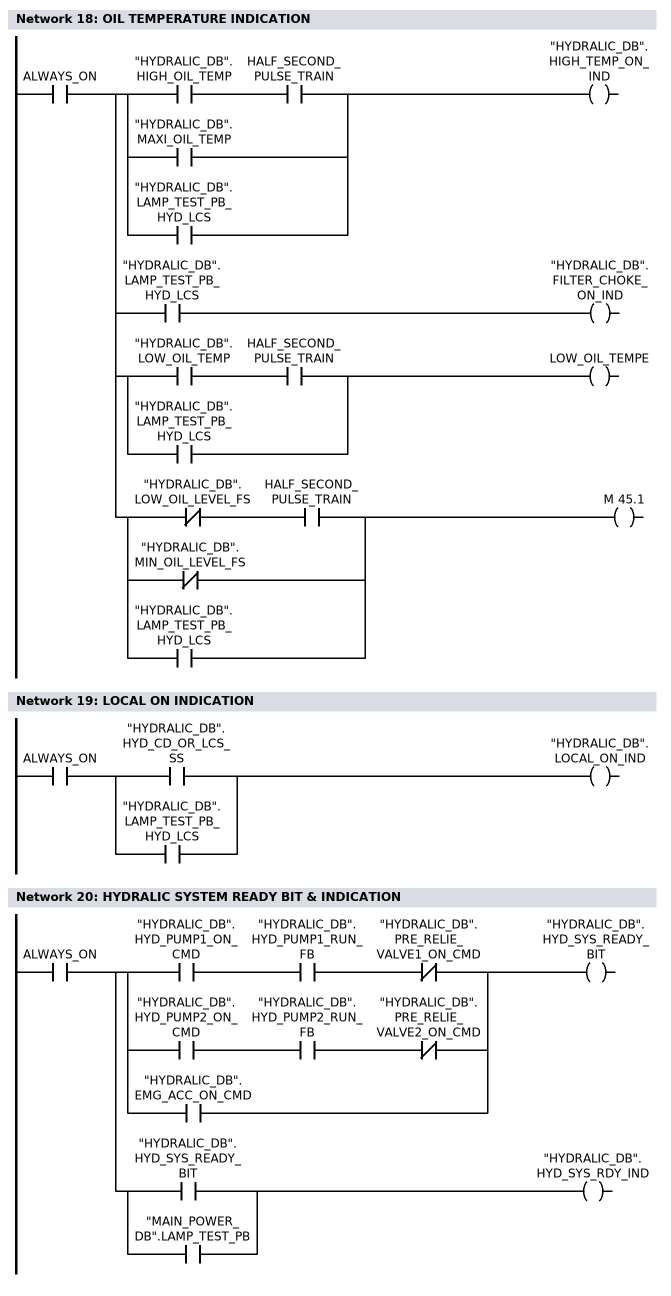
[picture p48: HYDRALIC_FUNCTION networks 18-20]
NETWORK
TITLE = OIL TEMPERATURE INDICATION
      A     "ALWAYS_ON";
      =     L 0.0;
      A     L 0.0;
      A(;
      A     "HYDRALIC_DB".HIGH_OIL_TEMP;
      A     "HALF_SECOND_PULSE_TRAIN";
      O     "HYDRALIC_DB".MAXI_OIL_TEMP;
      O     "HYDRALIC_DB".LAMP_TEST_PB_HYD_LCS;
      );
      =     "HYDRALIC_DB".HIGH_TEMP_ON_IND;
      A     L 0.0;
      A     "HYDRALIC_DB".LAMP_TEST_PB_HYD_LCS;
      =     "HYDRALIC_DB".FILTER_CHOKE_ON_IND;
      A     L 0.0;
      A(;
      A     "HYDRALIC_DB".LOW_OIL_TEMP;
      A     "HALF_SECOND_PULSE_TRAIN";
      O     "HYDRALIC_DB".LAMP_TEST_PB_HYD_LCS;
      );
      =     "LOW_OIL_TEMPE";
      A     L 0.0;
      A(;
      AN    "HYDRALIC_DB".LOW_OIL_LEVEL_FS;
      A     "HALF_SECOND_PULSE_TRAIN";
      ON    "HYDRALIC_DB".MIN_OIL_LEVEL_FS;
      O     "HYDRALIC_DB".LAMP_TEST_PB_HYD_LCS;
      );
      =     M 45.1;
NETWORK
TITLE = LOCAL ON INDICATION
      A     "ALWAYS_ON";
      A(;
      O     "HYDRALIC_DB".HYD_CD_OR_LCS_SS;
      O     "HYDRALIC_DB".LAMP_TEST_PB_HYD_LCS;
      );
      =     "HYDRALIC_DB".LOCAL_ON_IND;
NETWORK
TITLE = HYDRALIC SYSTEM READY BIT & INDICATION
      A     "ALWAYS_ON";
      =     L 0.0;
      A     L 0.0;
      A(;
      A     "HYDRALIC_DB".HYD_PUMP1_ON_CMD;
      A     "HYDRALIC_DB".HYD_PUMP1_RUN_FB;
      AN    "HYDRALIC_DB".PRE_RELIE_VALVE1_ON_CMD;
      O;
      A     "HYDRALIC_DB".HYD_PUMP2_ON_CMD;
      A     "HYDRALIC_DB".HYD_PUMP2_RUN_FB;
      AN    "HYDRALIC_DB".PRE_RELIE_VALVE2_ON_CMD;
      O     "HYDRALIC_DB".EMG_ACC_ON_CMD;
      );
      =     "HYDRALIC_DB".HYD_SYS_READY_BIT;
      A     L 0.0;
      A(;
      O     "HYDRALIC_DB".HYD_SYS_READY_BIT;
      O     "MAIN_POWER_DB".LAMP_TEST_PB;
      );
      =     "HYDRALIC_DB".HYD_SYS_RDY_IND;
END_FUNCTION

FUNCTION "TRAVEL_DRIVE" : VOID	// FC 8
AUTHOR : Arun_Ram
VERSION : 0.1
BEGIN
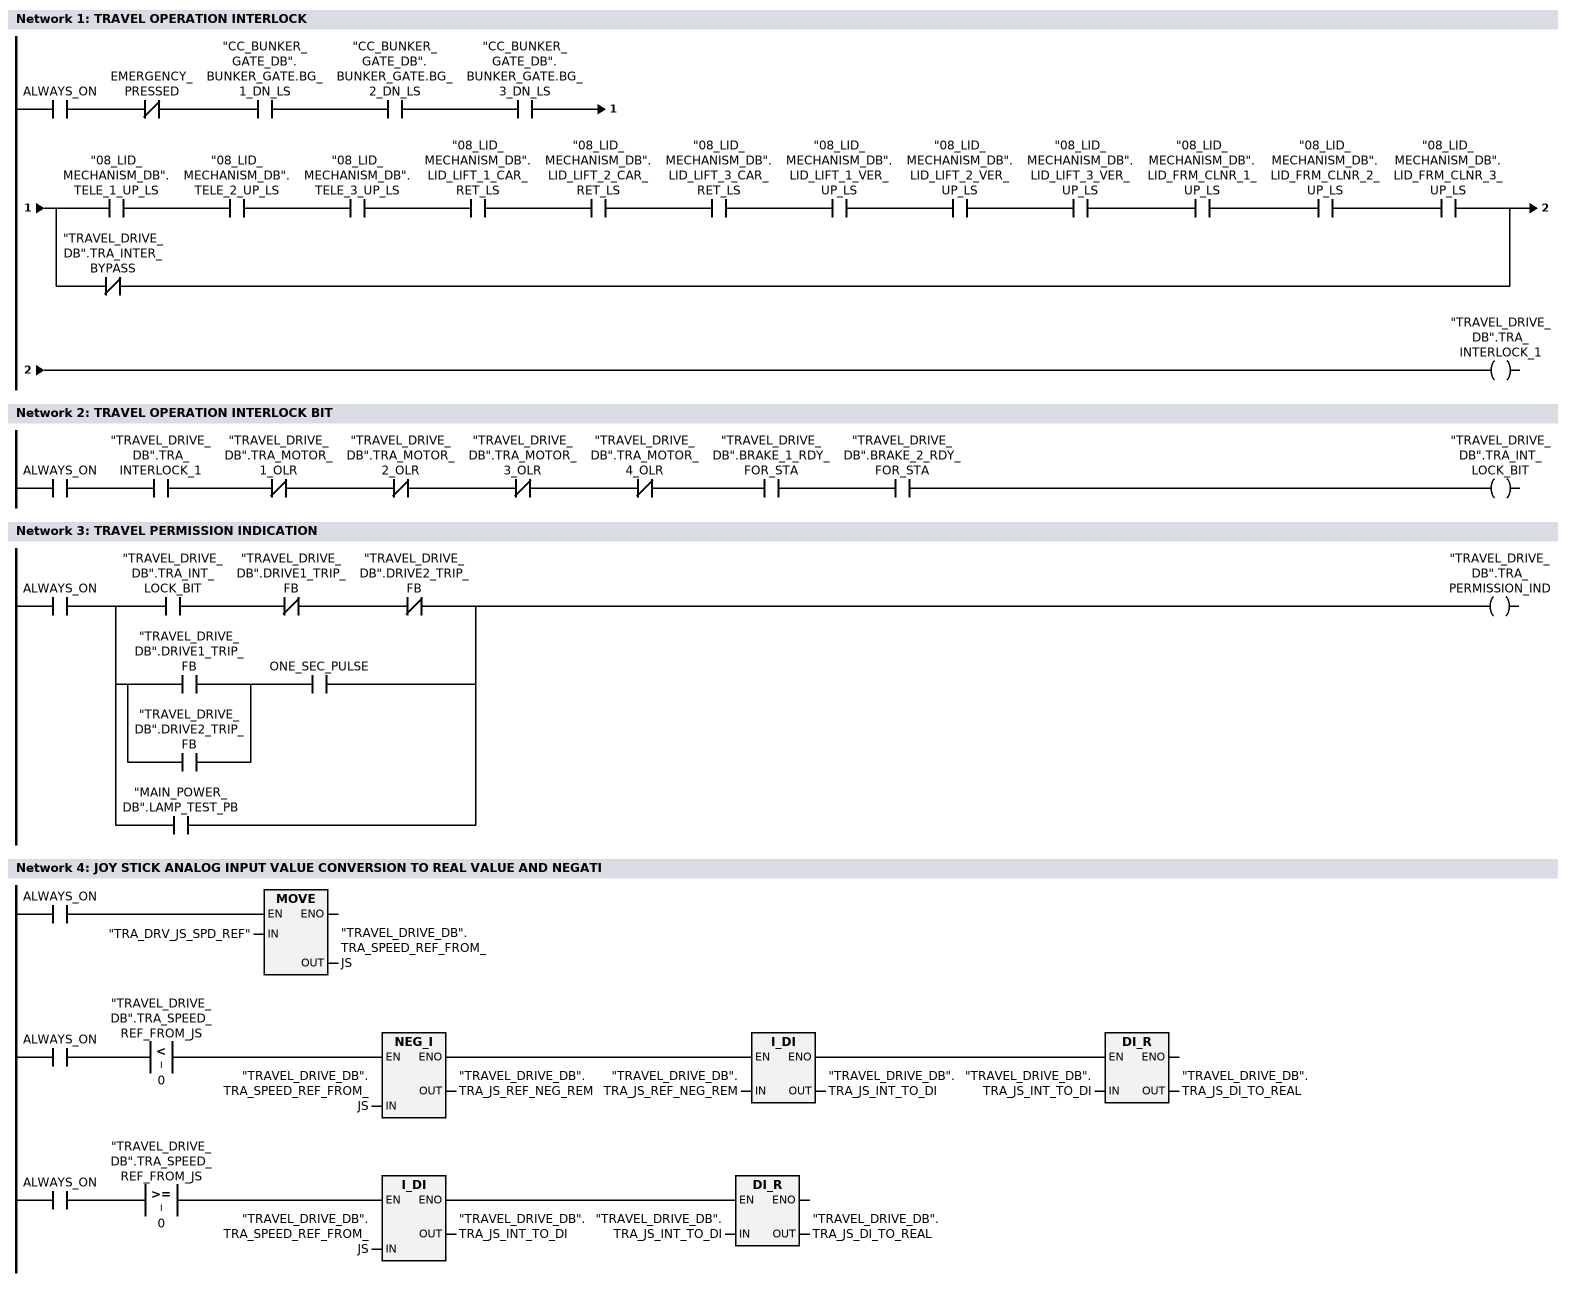
NETWORK
TITLE = TRAVEL OPERATION INTERLOCK
      A     "ALWAYS_ON";
      AN    "EMERGENCY_PRESSED";
      A     "CC_BUNKER_GATE_DB".BUNKER_GATE.BG_1_DN_LS;
      A     "CC_BUNKER_GATE_DB".BUNKER_GATE.BG_2_DN_LS;
      A     "CC_BUNKER_GATE_DB".BUNKER_GATE.BG_3_DN_LS;
      A(;
      A     "08_LID_MECHANISM_DB".TELE_1_UP_LS;
      A     "08_LID_MECHANISM_DB".TELE_2_UP_LS;
      A     "08_LID_MECHANISM_DB".TELE_3_UP_LS;
      A     "08_LID_MECHANISM_DB".LID_LIFT_1_CAR_RET_LS;
      A     "08_LID_MECHANISM_DB".LID_LIFT_2_CAR_RET_LS;
      A     "08_LID_MECHANISM_DB".LID_LIFT_3_CAR_RET_LS;
      A     "08_LID_MECHANISM_DB".LID_LIFT_1_VER_UP_LS;
      A     "08_LID_MECHANISM_DB".LID_LIFT_2_VER_UP_LS;
      A     "08_LID_MECHANISM_DB".LID_LIFT_3_VER_UP_LS;
      A     "08_LID_MECHANISM_DB".LID_FRM_CLNR_1_UP_LS;
      A     "08_LID_MECHANISM_DB".LID_FRM_CLNR_2_UP_LS;
      A     "08_LID_MECHANISM_DB".LID_FRM_CLNR_3_UP_LS;
      ON    "TRAVEL_DRIVE_DB".TRA_INTER_BYPASS;
      );
      =     "TRAVEL_DRIVE_DB".TRA_INTERLOCK_1;
NETWORK
TITLE = TRAVEL OPERATION INTERLOCK BIT
      A     "ALWAYS_ON";
      A     "TRAVEL_DRIVE_DB".TRA_INTERLOCK_1;
      AN    "TRAVEL_DRIVE_DB".TRA_MOTOR_1_OLR;
      AN    "TRAVEL_DRIVE_DB".TRA_MOTOR_2_OLR;
      AN    "TRAVEL_DRIVE_DB".TRA_MOTOR_3_OLR;
      AN    "TRAVEL_DRIVE_DB".TRA_MOTOR_4_OLR;
      A     "TRAVEL_DRIVE_DB".BRAKE_1_RDY_FOR_STA;
      A     "TRAVEL_DRIVE_DB".BRAKE_2_RDY_FOR_STA;
      =     "TRAVEL_DRIVE_DB".TRA_INT_LOCK_BIT;
NETWORK
TITLE = TRAVEL PERMISSION INDICATION
      A     "ALWAYS_ON";
      A(;
      A     "TRAVEL_DRIVE_DB".TRA_INT_LOCK_BIT;
      AN    "TRAVEL_DRIVE_DB".DRIVE1_TRIP_FB;
      AN    "TRAVEL_DRIVE_DB".DRIVE2_TRIP_FB;
      O;
      A(;
      O     "TRAVEL_DRIVE_DB".DRIVE1_TRIP_FB;
      O     "TRAVEL_DRIVE_DB".DRIVE2_TRIP_FB;
      );
      A     "ONE_SEC_PULSE";
      O     "MAIN_POWER_DB".LAMP_TEST_PB;
      );
      =     "TRAVEL_DRIVE_DB".TRA_PERMISSION_IND;
NETWORK
TITLE = JOY STICK ANALOG INPUT VALUE CONVERSION TO REAL VALUE AND NEGATI
//JOY STICK ANALOG INPUT VALUE CONVERTION TO REAL VALUE AND NEGATIVE TO POSITIVE 
//CONVERTION
      A     "ALWAYS_ON";
      =     L 0.0;
      A     L 0.0;
      JNB   _001;
      L     "TRA_DRV_JS_SPD_REF";
      T     "TRAVEL_DRIVE_DB".TRA_SPEED_REF_FROM_JS;
_001: NOP   0;
      A(;
      A(;
      A     L 0.0;
      A(;
      L     "TRAVEL_DRIVE_DB".TRA_SPEED_REF_FROM_JS;
      L     0;
      <I;
      );
      JNB   _002;
      L     "TRAVEL_DRIVE_DB".TRA_SPEED_REF_FROM_JS;
      NEGI;
      T     "TRAVEL_DRIVE_DB".TRA_JS_REF_NEG_REM;
      AN    OV;
      SAVE;
      CLR;
_002: A     BR;
      );
      JNB   _003;
      L     "TRAVEL_DRIVE_DB".TRA_JS_REF_NEG_REM;
      ITD;
      T     "TRAVEL_DRIVE_DB".TRA_JS_INT_TO_DI;
      SET;
      SAVE;
      CLR;
_003: A     BR;
      );
      JNB   _004;
      L     "TRAVEL_DRIVE_DB".TRA_JS_INT_TO_DI;
      DTR;
      T     "TRAVEL_DRIVE_DB".TRA_JS_DI_TO_REAL;
_004: NOP   0;
      A(;
      A     L 0.0;
      A(;
      L     "TRAVEL_DRIVE_DB".TRA_SPEED_REF_FROM_JS;
      L     0;
      >=I;
      );
      JNB   _005;
      L     "TRAVEL_DRIVE_DB".TRA_SPEED_REF_FROM_JS;
      ITD;
      T     "TRAVEL_DRIVE_DB".TRA_JS_INT_TO_DI;
      SET;
      SAVE;
      CLR;
_005: A     BR;
      );
      JNB   _006;
      L     "TRAVEL_DRIVE_DB".TRA_JS_INT_TO_DI;
      DTR;
      T     "TRAVEL_DRIVE_DB".TRA_JS_DI_TO_REAL;
_006: NOP   0;
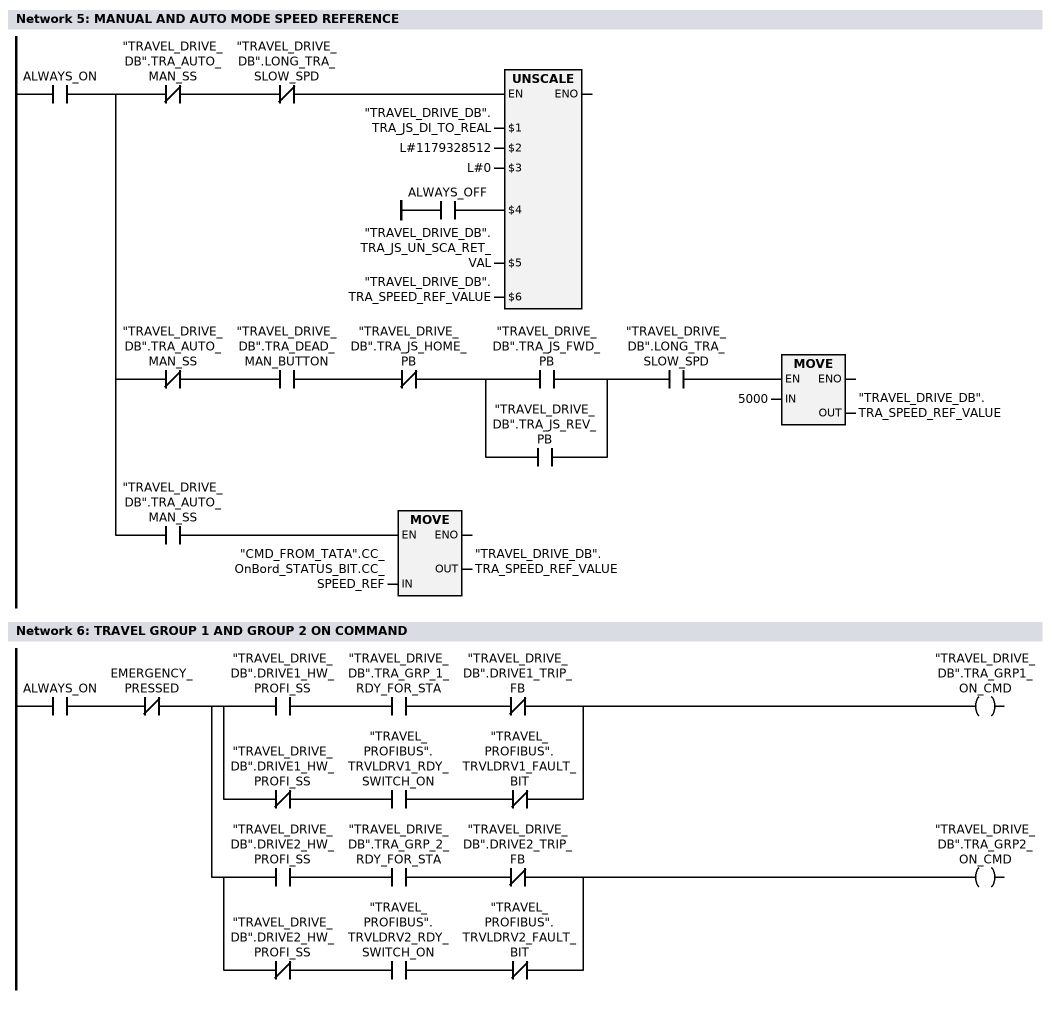
NETWORK
TITLE = MANUAL AND AUTO MODE SPEED REFERENCE
//JOY STICK ANALOG INPUT VALUE SCALLING WITH UNSCALLING BLOCK IN MANUAL MODE AND
//PROFIBUS SPEED REFERENCE VALUE TRANSFER IN AUTO MODE
//
      A     "ALWAYS_ON";
      =     L 0.0;
      A     "ALWAYS_OFF";
      =     L 0.1;
      BLD   103;
      A     L 0.0;
      AN    "TRAVEL_DRIVE_DB".TRA_AUTO_MAN_SS;
      AN    "TRAVEL_DRIVE_DB".LONG_TRA_SLOW_SPD;
      JNB   _007;
      CALL  "UNSCALE" (
           $1                       := "TRAVEL_DRIVE_DB".TRA_JS_DI_TO_REAL,
           $2                       := L#1179328512,
           $3                       := L#0,
           $4                       := L 0.1,
           $5                       := "TRAVEL_DRIVE_DB".TRA_JS_UN_SCA_RET_VAL,
           $6                       := "TRAVEL_DRIVE_DB".TRA_SPEED_REF_VALUE);
_007: NOP   0;
      A     L 0.0;
      AN    "TRAVEL_DRIVE_DB".TRA_AUTO_MAN_SS;
      A     "TRAVEL_DRIVE_DB".TRA_DEAD_MAN_BUTTON;
      AN    "TRAVEL_DRIVE_DB".TRA_JS_HOME_PB;
      A(;
      O     "TRAVEL_DRIVE_DB".TRA_JS_FWD_PB;
      O     "TRAVEL_DRIVE_DB".TRA_JS_REV_PB;
      );
      A     "TRAVEL_DRIVE_DB".LONG_TRA_SLOW_SPD;
      JNB   _008;
      L     5000;
      T     "TRAVEL_DRIVE_DB".TRA_SPEED_REF_VALUE;
_008: NOP   0;
      A     L 0.0;
      A     "TRAVEL_DRIVE_DB".TRA_AUTO_MAN_SS;
      JNB   _009;
      L     "CMD_FROM_TATA".CC_OnBord_STATUS_BIT.CC_SPEED_REF;
      T     "TRAVEL_DRIVE_DB".TRA_SPEED_REF_VALUE;
_009: NOP   0;
NETWORK
TITLE = TRAVEL GROUP 1 AND GROUP 2 ON COMMAND
      A     "ALWAYS_ON";
      AN    "EMERGENCY_PRESSED";
      =     L 0.0;
      A     L 0.0;
      A(;
      A     "TRAVEL_DRIVE_DB".DRIVE1_HW_PROFI_SS;
      A     "TRAVEL_DRIVE_DB".TRA_GRP_1_RDY_FOR_STA;
      AN    "TRAVEL_DRIVE_DB".DRIVE1_TRIP_FB;
      O;
      AN    "TRAVEL_DRIVE_DB".DRIVE1_HW_PROFI_SS;
      A     "TRAVEL_PROFIBUS".TRVLDRV1_RDY_SWITCH_ON;
      AN    "TRAVEL_PROFIBUS".TRVLDRV1_FAULT_BIT;
      );
      =     "TRAVEL_DRIVE_DB".TRA_GRP1_ON_CMD;
      A     L 0.0;
      A(;
      A     "TRAVEL_DRIVE_DB".DRIVE2_HW_PROFI_SS;
      A     "TRAVEL_DRIVE_DB".TRA_GRP_2_RDY_FOR_STA;
      AN    "TRAVEL_DRIVE_DB".DRIVE2_TRIP_FB;
      O;
      AN    "TRAVEL_DRIVE_DB".DRIVE2_HW_PROFI_SS;
      A     "TRAVEL_PROFIBUS".TRVLDRV2_RDY_SWITCH_ON;
      AN    "TRAVEL_PROFIBUS".TRVLDRV2_FAULT_BIT;
      );
      =     "TRAVEL_DRIVE_DB".TRA_GRP2_ON_CMD;
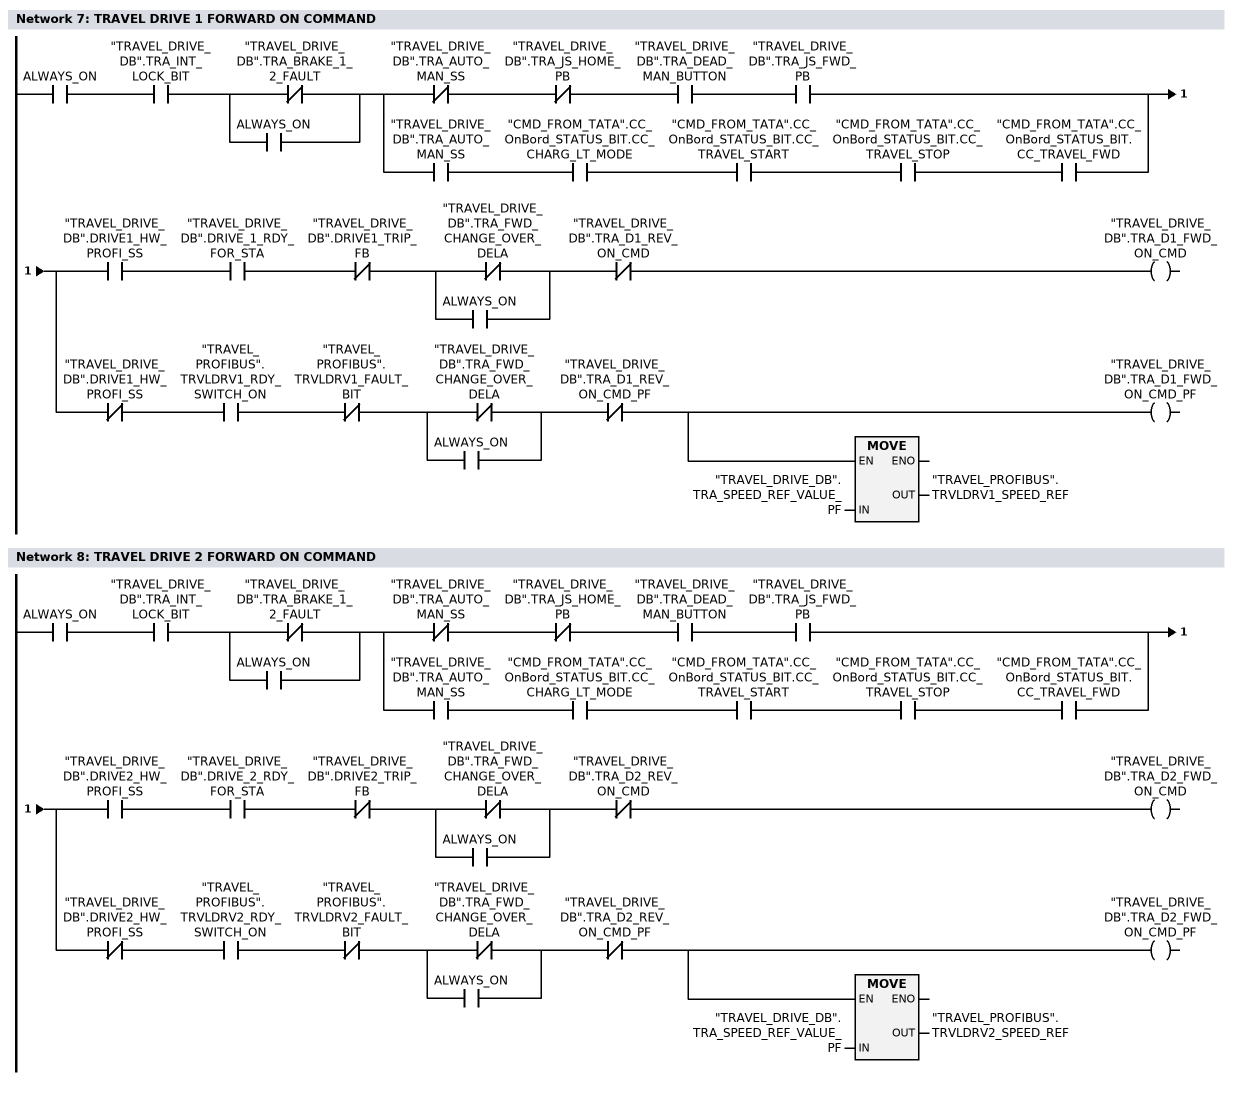
NETWORK
TITLE = TRAVEL DRIVE 1 FORWARD ON COMMAND
      A     "ALWAYS_ON";
      A     "TRAVEL_DRIVE_DB".TRA_INT_LOCK_BIT;
      A(;
      ON    "TRAVEL_DRIVE_DB".TRA_BRAKE_1_2_FAULT;
      O     "ALWAYS_ON";
      );
      A(;
      AN    "TRAVEL_DRIVE_DB".TRA_AUTO_MAN_SS;
      AN    "TRAVEL_DRIVE_DB".TRA_JS_HOME_PB;
      A     "TRAVEL_DRIVE_DB".TRA_DEAD_MAN_BUTTON;
      A     "TRAVEL_DRIVE_DB".TRA_JS_FWD_PB;
      O;
      A     "TRAVEL_DRIVE_DB".TRA_AUTO_MAN_SS;
      A     "CMD_FROM_TATA".CC_OnBord_STATUS_BIT.CC_CHARG_LT_MODE;
      A     "CMD_FROM_TATA".CC_OnBord_STATUS_BIT.CC_TRAVEL_START;
      A     "CMD_FROM_TATA".CC_OnBord_STATUS_BIT.CC_TRAVEL_STOP;
      A     "CMD_FROM_TATA".CC_OnBord_STATUS_BIT.CC_TRAVEL_FWD;
      );
      =     L 0.0;
      A     L 0.0;
      A     "TRAVEL_DRIVE_DB".DRIVE1_HW_PROFI_SS;
      A     "TRAVEL_DRIVE_DB".DRIVE_1_RDY_FOR_STA;
      AN    "TRAVEL_DRIVE_DB".DRIVE1_TRIP_FB;
      A(;
      ON    "TRAVEL_DRIVE_DB".TRA_FWD_CHANGE_OVER_DELA;
      O     "ALWAYS_ON";
      );
      AN    "TRAVEL_DRIVE_DB".TRA_D1_REV_ON_CMD;
      =     "TRAVEL_DRIVE_DB".TRA_D1_FWD_ON_CMD;
      A     L 0.0;
      AN    "TRAVEL_DRIVE_DB".DRIVE1_HW_PROFI_SS;
      A     "TRAVEL_PROFIBUS".TRVLDRV1_RDY_SWITCH_ON;
      AN    "TRAVEL_PROFIBUS".TRVLDRV1_FAULT_BIT;
      A(;
      ON    "TRAVEL_DRIVE_DB".TRA_FWD_CHANGE_OVER_DELA;
      O     "ALWAYS_ON";
      );
      AN    "TRAVEL_DRIVE_DB".TRA_D1_REV_ON_CMD_PF;
      =     L 0.1;
      A     L 0.1;
      BLD   102;
      =     "TRAVEL_DRIVE_DB".TRA_D1_FWD_ON_CMD_PF;
      A     L 0.1;
      JNB   _00a;
      L     "TRAVEL_DRIVE_DB".TRA_SPEED_REF_VALUE_PF;
      T     "TRAVEL_PROFIBUS".TRVLDRV1_SPEED_REF;
_00a: NOP   0;
NETWORK
TITLE = TRAVEL DRIVE 2 FORWARD ON COMMAND
      A     "ALWAYS_ON";
      A     "TRAVEL_DRIVE_DB".TRA_INT_LOCK_BIT;
      A(;
      ON    "TRAVEL_DRIVE_DB".TRA_BRAKE_1_2_FAULT;
      O     "ALWAYS_ON";
      );
      A(;
      AN    "TRAVEL_DRIVE_DB".TRA_AUTO_MAN_SS;
      AN    "TRAVEL_DRIVE_DB".TRA_JS_HOME_PB;
      A     "TRAVEL_DRIVE_DB".TRA_DEAD_MAN_BUTTON;
      A     "TRAVEL_DRIVE_DB".TRA_JS_FWD_PB;
      O;
      A     "TRAVEL_DRIVE_DB".TRA_AUTO_MAN_SS;
      A     "CMD_FROM_TATA".CC_OnBord_STATUS_BIT.CC_CHARG_LT_MODE;
      A     "CMD_FROM_TATA".CC_OnBord_STATUS_BIT.CC_TRAVEL_START;
      A     "CMD_FROM_TATA".CC_OnBord_STATUS_BIT.CC_TRAVEL_STOP;
      A     "CMD_FROM_TATA".CC_OnBord_STATUS_BIT.CC_TRAVEL_FWD;
      );
      =     L 0.0;
      A     L 0.0;
      A     "TRAVEL_DRIVE_DB".DRIVE2_HW_PROFI_SS;
      A     "TRAVEL_DRIVE_DB".DRIVE_2_RDY_FOR_STA;
      AN    "TRAVEL_DRIVE_DB".DRIVE2_TRIP_FB;
      A(;
      ON    "TRAVEL_DRIVE_DB".TRA_FWD_CHANGE_OVER_DELA;
      O     "ALWAYS_ON";
      );
      AN    "TRAVEL_DRIVE_DB".TRA_D2_REV_ON_CMD;
      =     "TRAVEL_DRIVE_DB".TRA_D2_FWD_ON_CMD;
      A     L 0.0;
      AN    "TRAVEL_DRIVE_DB".DRIVE2_HW_PROFI_SS;
      A     "TRAVEL_PROFIBUS".TRVLDRV2_RDY_SWITCH_ON;
      AN    "TRAVEL_PROFIBUS".TRVLDRV2_FAULT_BIT;
      A(;
      ON    "TRAVEL_DRIVE_DB".TRA_FWD_CHANGE_OVER_DELA;
      O     "ALWAYS_ON";
      );
      AN    "TRAVEL_DRIVE_DB".TRA_D2_REV_ON_CMD_PF;
      =     L 0.1;
      A     L 0.1;
      BLD   102;
      =     "TRAVEL_DRIVE_DB".TRA_D2_FWD_ON_CMD_PF;
      A     L 0.1;
      JNB   _00b;
      L     "TRAVEL_DRIVE_DB".TRA_SPEED_REF_VALUE_PF;
      T     "TRAVEL_PROFIBUS".TRVLDRV2_SPEED_REF;
_00b: NOP   0;
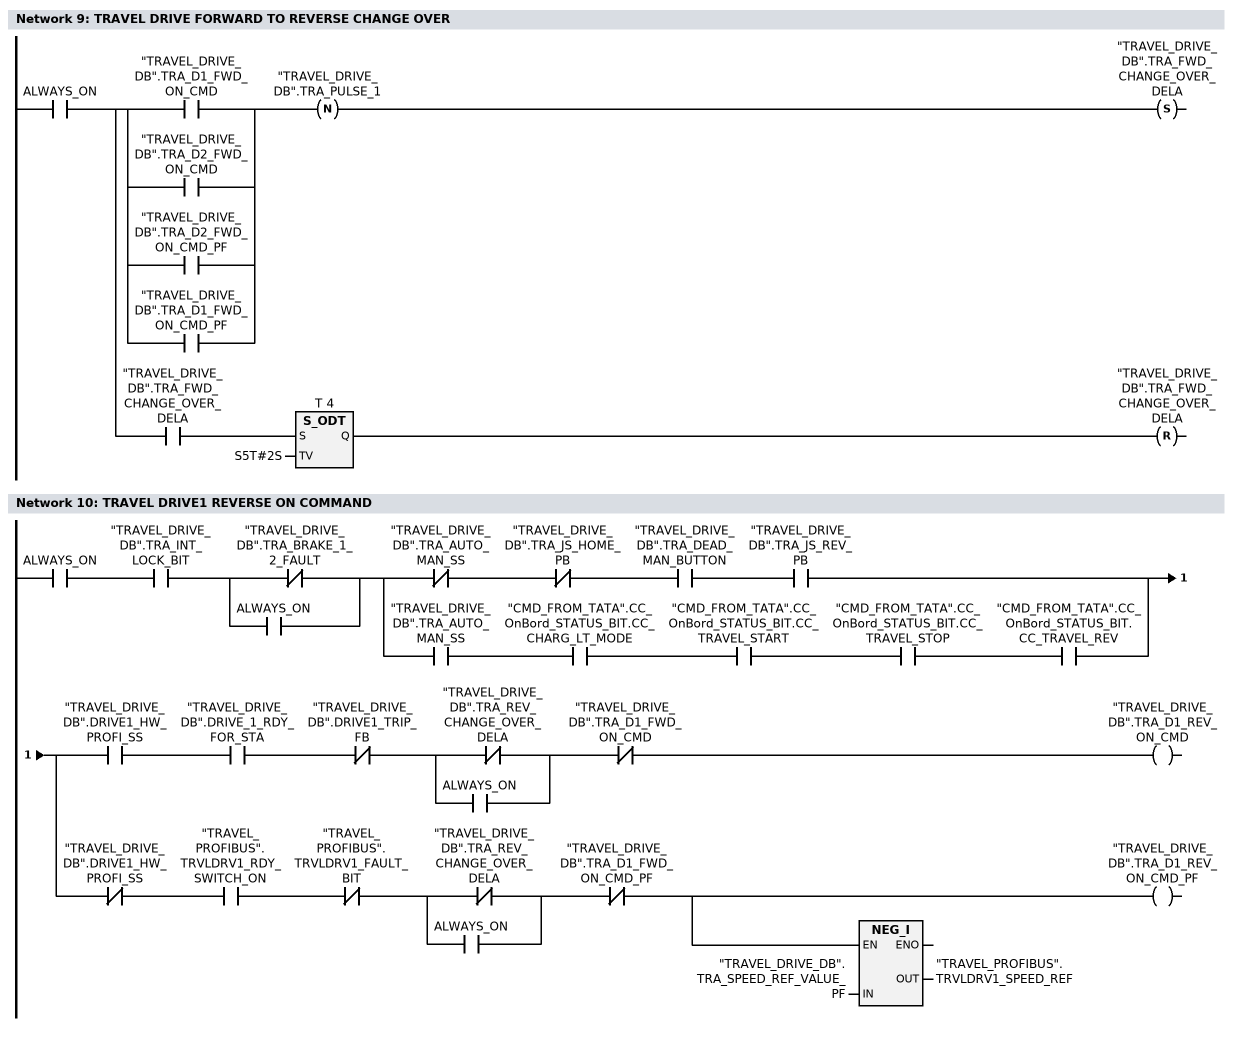
NETWORK
TITLE = TRAVEL DRIVE FORWARD TO REVERSE CHANGE OVER
      A     "ALWAYS_ON";
      =     L 0.0;
      A     L 0.0;
      A(;
      O     "TRAVEL_DRIVE_DB".TRA_D1_FWD_ON_CMD;
      O     "TRAVEL_DRIVE_DB".TRA_D2_FWD_ON_CMD;
      O     "TRAVEL_DRIVE_DB".TRA_D2_FWD_ON_CMD_PF;
      O     "TRAVEL_DRIVE_DB".TRA_D1_FWD_ON_CMD_PF;
      );
      FN    "TRAVEL_DRIVE_DB".TRA_PULSE_1;
      S     "TRAVEL_DRIVE_DB".TRA_FWD_CHANGE_OVER_DELA;
      A     L 0.0;
      A     "TRAVEL_DRIVE_DB".TRA_FWD_CHANGE_OVER_DELA;
      L     S5T#2S;
      SD    T 4;
      NOP   0;
      NOP   0;
      NOP   0;
      A     T 4;
      R     "TRAVEL_DRIVE_DB".TRA_FWD_CHANGE_OVER_DELA;
NETWORK
TITLE = TRAVEL DRIVE1 REVERSE ON COMMAND
      A     "ALWAYS_ON";
      A     "TRAVEL_DRIVE_DB".TRA_INT_LOCK_BIT;
      A(;
      ON    "TRAVEL_DRIVE_DB".TRA_BRAKE_1_2_FAULT;
      O     "ALWAYS_ON";
      );
      A(;
      AN    "TRAVEL_DRIVE_DB".TRA_AUTO_MAN_SS;
      AN    "TRAVEL_DRIVE_DB".TRA_JS_HOME_PB;
      A     "TRAVEL_DRIVE_DB".TRA_DEAD_MAN_BUTTON;
      A     "TRAVEL_DRIVE_DB".TRA_JS_REV_PB;
      O;
      A     "TRAVEL_DRIVE_DB".TRA_AUTO_MAN_SS;
      A     "CMD_FROM_TATA".CC_OnBord_STATUS_BIT.CC_CHARG_LT_MODE;
      A     "CMD_FROM_TATA".CC_OnBord_STATUS_BIT.CC_TRAVEL_START;
      A     "CMD_FROM_TATA".CC_OnBord_STATUS_BIT.CC_TRAVEL_STOP;
      A     "CMD_FROM_TATA".CC_OnBord_STATUS_BIT.CC_TRAVEL_REV;
      );
      =     L 0.0;
      A     L 0.0;
      A     "TRAVEL_DRIVE_DB".DRIVE1_HW_PROFI_SS;
      A     "TRAVEL_DRIVE_DB".DRIVE_1_RDY_FOR_STA;
      AN    "TRAVEL_DRIVE_DB".DRIVE1_TRIP_FB;
      A(;
      ON    "TRAVEL_DRIVE_DB".TRA_REV_CHANGE_OVER_DELA;
      O     "ALWAYS_ON";
      );
      AN    "TRAVEL_DRIVE_DB".TRA_D1_FWD_ON_CMD;
      =     "TRAVEL_DRIVE_DB".TRA_D1_REV_ON_CMD;
      A     L 0.0;
      AN    "TRAVEL_DRIVE_DB".DRIVE1_HW_PROFI_SS;
      A     "TRAVEL_PROFIBUS".TRVLDRV1_RDY_SWITCH_ON;
      AN    "TRAVEL_PROFIBUS".TRVLDRV1_FAULT_BIT;
      A(;
      ON    "TRAVEL_DRIVE_DB".TRA_REV_CHANGE_OVER_DELA;
      O     "ALWAYS_ON";
      );
      AN    "TRAVEL_DRIVE_DB".TRA_D1_FWD_ON_CMD_PF;
      =     L 0.1;
      A     L 0.1;
      BLD   102;
      =     "TRAVEL_DRIVE_DB".TRA_D1_REV_ON_CMD_PF;
      A     L 0.1;
      JNB   _00c;
      L     "TRAVEL_DRIVE_DB".TRA_SPEED_REF_VALUE_PF;
      NEGI;
      T     "TRAVEL_PROFIBUS".TRVLDRV1_SPEED_REF;
_00c: NOP   0;
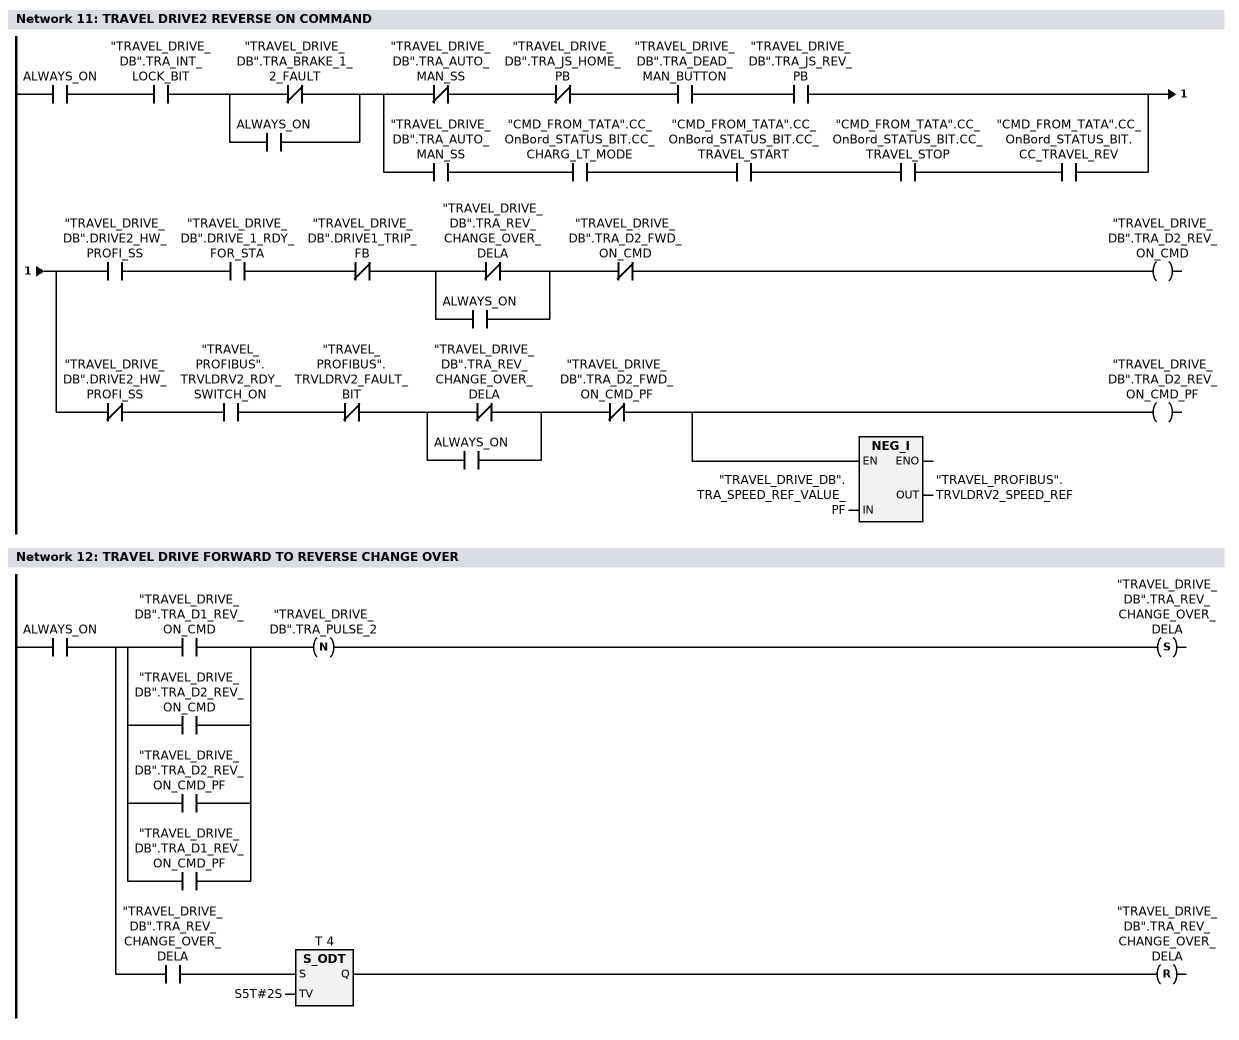
NETWORK
TITLE = TRAVEL DRIVE2 REVERSE ON COMMAND
      A     "ALWAYS_ON";
      A     "TRAVEL_DRIVE_DB".TRA_INT_LOCK_BIT;
      A(;
      ON    "TRAVEL_DRIVE_DB".TRA_BRAKE_1_2_FAULT;
      O     "ALWAYS_ON";
      );
      A(;
      AN    "TRAVEL_DRIVE_DB".TRA_AUTO_MAN_SS;
      AN    "TRAVEL_DRIVE_DB".TRA_JS_HOME_PB;
      A     "TRAVEL_DRIVE_DB".TRA_DEAD_MAN_BUTTON;
      A     "TRAVEL_DRIVE_DB".TRA_JS_REV_PB;
      O;
      A     "TRAVEL_DRIVE_DB".TRA_AUTO_MAN_SS;
      A     "CMD_FROM_TATA".CC_OnBord_STATUS_BIT.CC_CHARG_LT_MODE;
      A     "CMD_FROM_TATA".CC_OnBord_STATUS_BIT.CC_TRAVEL_START;
      A     "CMD_FROM_TATA".CC_OnBord_STATUS_BIT.CC_TRAVEL_STOP;
      A     "CMD_FROM_TATA".CC_OnBord_STATUS_BIT.CC_TRAVEL_REV;
      );
      =     L 0.0;
      A     L 0.0;
      A     "TRAVEL_DRIVE_DB".DRIVE2_HW_PROFI_SS;
      A     "TRAVEL_DRIVE_DB".DRIVE_1_RDY_FOR_STA;
      AN    "TRAVEL_DRIVE_DB".DRIVE1_TRIP_FB;
      A(;
      ON    "TRAVEL_DRIVE_DB".TRA_REV_CHANGE_OVER_DELA;
      O     "ALWAYS_ON";
      );
      AN    "TRAVEL_DRIVE_DB".TRA_D2_FWD_ON_CMD;
      =     "TRAVEL_DRIVE_DB".TRA_D2_REV_ON_CMD;
      A     L 0.0;
      AN    "TRAVEL_DRIVE_DB".DRIVE2_HW_PROFI_SS;
      A     "TRAVEL_PROFIBUS".TRVLDRV2_RDY_SWITCH_ON;
      AN    "TRAVEL_PROFIBUS".TRVLDRV2_FAULT_BIT;
      A(;
      ON    "TRAVEL_DRIVE_DB".TRA_REV_CHANGE_OVER_DELA;
      O     "ALWAYS_ON";
      );
      AN    "TRAVEL_DRIVE_DB".TRA_D2_FWD_ON_CMD_PF;
      =     L 0.1;
      A     L 0.1;
      BLD   102;
      =     "TRAVEL_DRIVE_DB".TRA_D2_REV_ON_CMD_PF;
      A     L 0.1;
      JNB   _00d;
      L     "TRAVEL_DRIVE_DB".TRA_SPEED_REF_VALUE_PF;
      NEGI;
      T     "TRAVEL_PROFIBUS".TRVLDRV2_SPEED_REF;
_00d: NOP   0;
NETWORK
TITLE = TRAVEL DRIVE FORWARD TO REVERSE CHANGE OVER
      A     "ALWAYS_ON";
      =     L 0.0;
      A     L 0.0;
      A(;
      O     "TRAVEL_DRIVE_DB".TRA_D1_REV_ON_CMD;
      O     "TRAVEL_DRIVE_DB".TRA_D2_REV_ON_CMD;
      O     "TRAVEL_DRIVE_DB".TRA_D2_REV_ON_CMD_PF;
      O     "TRAVEL_DRIVE_DB".TRA_D1_REV_ON_CMD_PF;
      );
      FN    "TRAVEL_DRIVE_DB".TRA_PULSE_2;
      S     "TRAVEL_DRIVE_DB".TRA_REV_CHANGE_OVER_DELA;
      A     L 0.0;
      A     "TRAVEL_DRIVE_DB".TRA_REV_CHANGE_OVER_DELA;
      L     S5T#2S;
      SD    T 4;
      NOP   0;
      NOP   0;
      NOP   0;
      A     T 4;
      R     "TRAVEL_DRIVE_DB".TRA_REV_CHANGE_OVER_DELA;
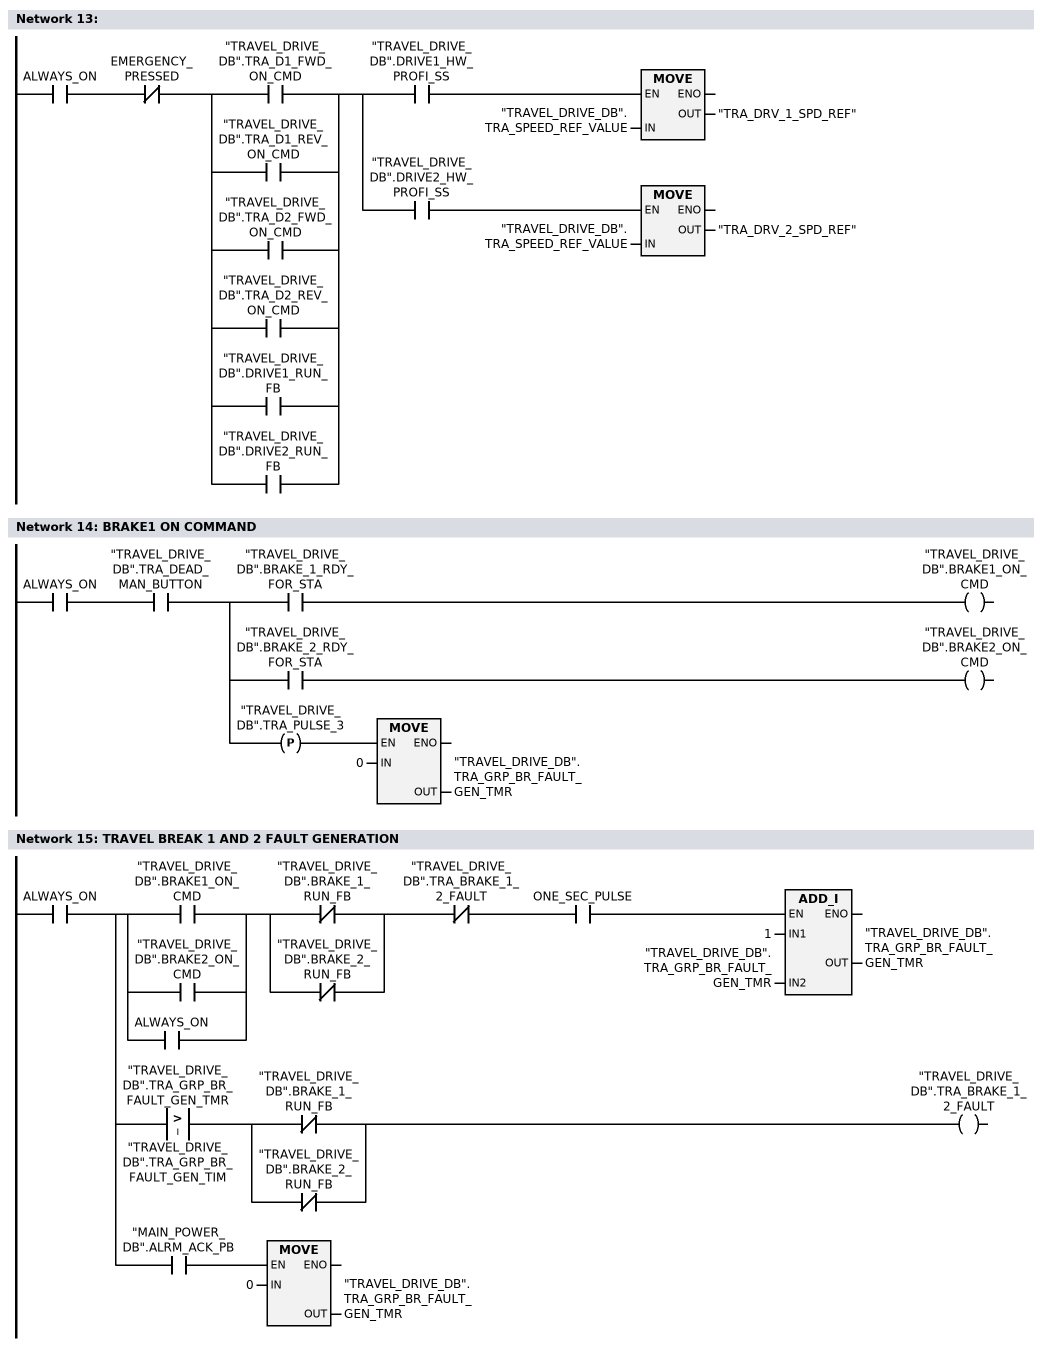
NETWORK
TITLE =
      A     "ALWAYS_ON";
      AN    "EMERGENCY_PRESSED";
      A(;
      O     "TRAVEL_DRIVE_DB".TRA_D1_FWD_ON_CMD;
      O     "TRAVEL_DRIVE_DB".TRA_D1_REV_ON_CMD;
      O     "TRAVEL_DRIVE_DB".TRA_D2_FWD_ON_CMD;
      O     "TRAVEL_DRIVE_DB".TRA_D2_REV_ON_CMD;
      O     "TRAVEL_DRIVE_DB".DRIVE1_RUN_FB;
      O     "TRAVEL_DRIVE_DB".DRIVE2_RUN_FB;
      );
      =     L 0.0;
      A     L 0.0;
      A     "TRAVEL_DRIVE_DB".DRIVE1_HW_PROFI_SS;
      JNB   _00e;
      L     "TRAVEL_DRIVE_DB".TRA_SPEED_REF_VALUE;
      T     "TRA_DRV_1_SPD_REF";
_00e: NOP   0;
      A     L 0.0;
      A     "TRAVEL_DRIVE_DB".DRIVE2_HW_PROFI_SS;
      JNB   _00f;
      L     "TRAVEL_DRIVE_DB".TRA_SPEED_REF_VALUE;
      T     "TRA_DRV_2_SPD_REF";
_00f: NOP   0;
NETWORK
TITLE = BRAKE1 ON COMMAND
      A     "ALWAYS_ON";
      A     "TRAVEL_DRIVE_DB".TRA_DEAD_MAN_BUTTON;
      =     L 0.0;
      A     L 0.0;
      A     "TRAVEL_DRIVE_DB".BRAKE_1_RDY_FOR_STA;
      =     "TRAVEL_DRIVE_DB".BRAKE1_ON_CMD;
      A     L 0.0;
      A     "TRAVEL_DRIVE_DB".BRAKE_2_RDY_FOR_STA;
      =     "TRAVEL_DRIVE_DB".BRAKE2_ON_CMD;
      A     L 0.0;
      FP    "TRAVEL_DRIVE_DB".TRA_PULSE_3;
      JNB   _010;
      L     0;
      T     "TRAVEL_DRIVE_DB".TRA_GRP_BR_FAULT_GEN_TMR;
_010: NOP   0;
NETWORK
TITLE = TRAVEL BREAK 1 AND 2 FAULT GENERATION
      A     "ALWAYS_ON";
      =     L 0.0;
      A     L 0.0;
      A(;
      O     "TRAVEL_DRIVE_DB".BRAKE1_ON_CMD;
      O     "TRAVEL_DRIVE_DB".BRAKE2_ON_CMD;
      O     "ALWAYS_ON";
      );
      A(;
      ON    "TRAVEL_DRIVE_DB".BRAKE_1_RUN_FB;
      ON    "TRAVEL_DRIVE_DB".BRAKE_2_RUN_FB;
      );
      AN    "TRAVEL_DRIVE_DB".TRA_BRAKE_1_2_FAULT;
      A     "ONE_SEC_PULSE";
      JNB   _011;
      L     1;
      L     "TRAVEL_DRIVE_DB".TRA_GRP_BR_FAULT_GEN_TMR;
      +I;
      T     "TRAVEL_DRIVE_DB".TRA_GRP_BR_FAULT_GEN_TMR;
_011: NOP   0;
      A     L 0.0;
      A(;
      L     "TRAVEL_DRIVE_DB".TRA_GRP_BR_FAULT_GEN_TMR;
      L     "TRAVEL_DRIVE_DB".TRA_GRP_BR_FAULT_GEN_TIM;
      >I;
      );
      A(;
      ON    "TRAVEL_DRIVE_DB".BRAKE_1_RUN_FB;
      ON    "TRAVEL_DRIVE_DB".BRAKE_2_RUN_FB;
      );
      =     "TRAVEL_DRIVE_DB".TRA_BRAKE_1_2_FAULT;
      A     L 0.0;
      A     "MAIN_POWER_DB".ALRM_ACK_PB;
      JNB   _012;
      L     0;
      T     "TRAVEL_DRIVE_DB".TRA_GRP_BR_FAULT_GEN_TMR;
_012: NOP   0;
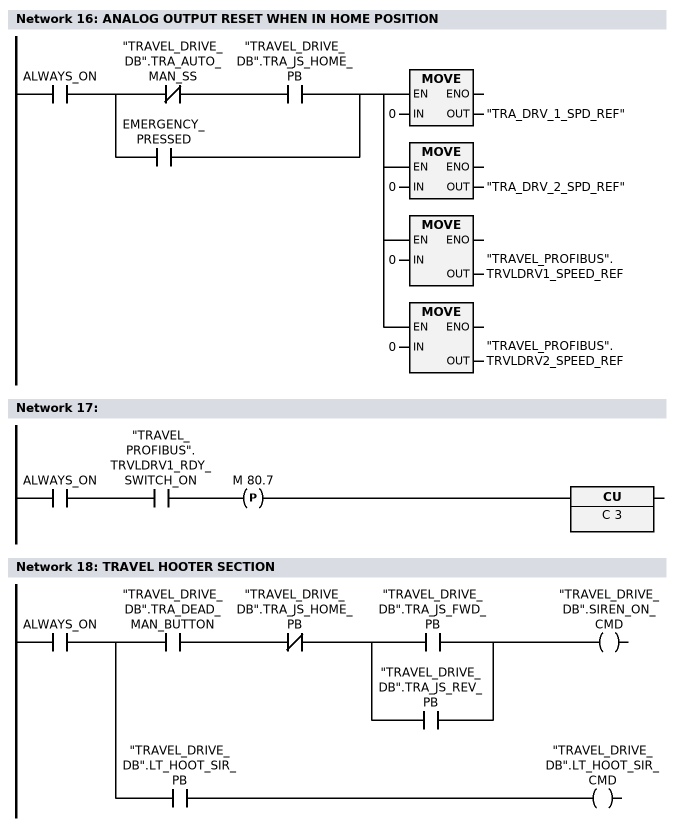
NETWORK
TITLE = ANALOG OUTPUT RESET WHEN IN HOME POSITION
      A     "ALWAYS_ON";
      A(;
      AN    "TRAVEL_DRIVE_DB".TRA_AUTO_MAN_SS;
      A     "TRAVEL_DRIVE_DB".TRA_JS_HOME_PB;
      O     "EMERGENCY_PRESSED";
      );
      =     L 0.0;
      A     L 0.0;
      JNB   _013;
      L     0;
      T     "TRA_DRV_1_SPD_REF";
_013: NOP   0;
      A     L 0.0;
      JNB   _014;
      L     0;
      T     "TRA_DRV_2_SPD_REF";
_014: NOP   0;
      A     L 0.0;
      JNB   _015;
      L     0;
      T     "TRAVEL_PROFIBUS".TRVLDRV1_SPEED_REF;
_015: NOP   0;
      A     L 0.0;
      JNB   _016;
      L     0;
      T     "TRAVEL_PROFIBUS".TRVLDRV2_SPEED_REF;
_016: NOP   0;
NETWORK
TITLE =
      A     "ALWAYS_ON";
      A     "TRAVEL_PROFIBUS".TRVLDRV1_RDY_SWITCH_ON;
      FP    M 80.7;
      CU    C 3;
      BLD   101;
      NOP   0;
      NOP   0;
      NOP   0;
      NOP   0;
      NOP   0;
      NOP   0;
NETWORK
TITLE = TRAVEL HOOTER SECTION
      A     "ALWAYS_ON";
      =     L 0.0;
      A     L 0.0;
      A     "TRAVEL_DRIVE_DB".TRA_DEAD_MAN_BUTTON;
      AN    "TRAVEL_DRIVE_DB".TRA_JS_HOME_PB;
      A(;
      O     "TRAVEL_DRIVE_DB".TRA_JS_FWD_PB;
      O     "TRAVEL_DRIVE_DB".TRA_JS_REV_PB;
      );
      =     "TRAVEL_DRIVE_DB".SIREN_ON_CMD;
      A     L 0.0;
      A     "TRAVEL_DRIVE_DB".LT_HOOT_SIR_PB;
      =     "TRAVEL_DRIVE_DB".LT_HOOT_SIR_CMD;
END_FUNCTION

FUNCTION "BUNKER_GATE" : VOID	// FC 9
AUTHOR : Arun
VERSION : 0.1
BEGIN
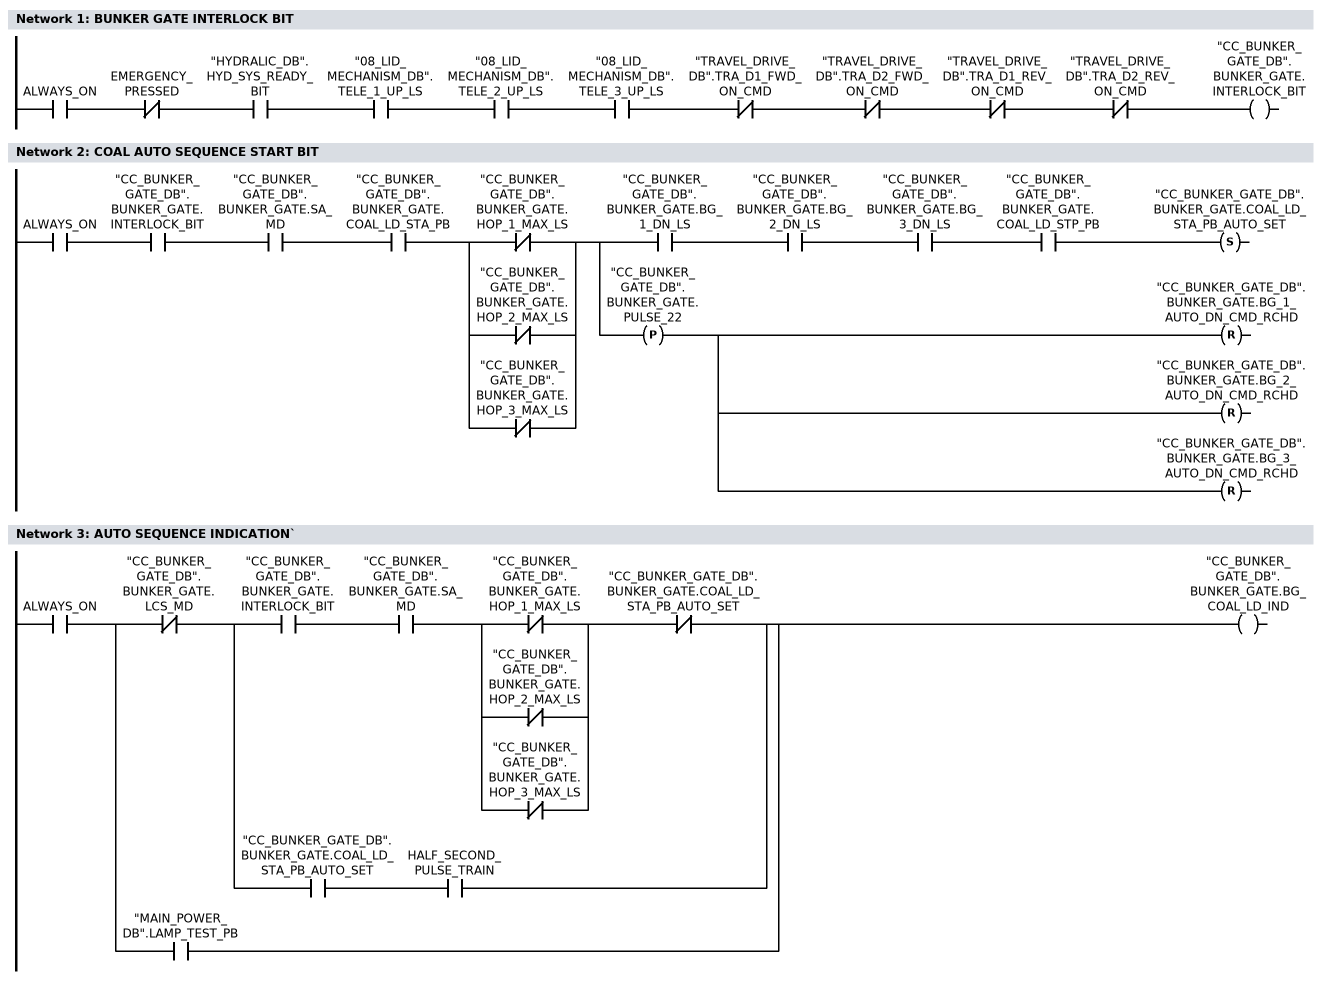
NETWORK
TITLE = BUNKER GATE INTERLOCK BIT
      A     "ALWAYS_ON";
      AN    "EMERGENCY_PRESSED";
      A     "HYDRALIC_DB".HYD_SYS_READY_BIT;
      A     "08_LID_MECHANISM_DB".TELE_1_UP_LS;
      A     "08_LID_MECHANISM_DB".TELE_2_UP_LS;
      A     "08_LID_MECHANISM_DB".TELE_3_UP_LS;
      AN    "TRAVEL_DRIVE_DB".TRA_D1_FWD_ON_CMD;
      AN    "TRAVEL_DRIVE_DB".TRA_D2_FWD_ON_CMD;
      AN    "TRAVEL_DRIVE_DB".TRA_D1_REV_ON_CMD;
      AN    "TRAVEL_DRIVE_DB".TRA_D2_REV_ON_CMD;
      =     "CC_BUNKER_GATE_DB".BUNKER_GATE.INTERLOCK_BIT;
NETWORK
TITLE = COAL AUTO SEQUENCE START BIT
      A     "ALWAYS_ON";
      A     "CC_BUNKER_GATE_DB".BUNKER_GATE.INTERLOCK_BIT;
      A     "CC_BUNKER_GATE_DB".BUNKER_GATE.SA_MD;
      A     "CC_BUNKER_GATE_DB".BUNKER_GATE.COAL_LD_STA_PB;
      A(;
      ON    "CC_BUNKER_GATE_DB".BUNKER_GATE.HOP_1_MAX_LS;
      ON    "CC_BUNKER_GATE_DB".BUNKER_GATE.HOP_2_MAX_LS;
      ON    "CC_BUNKER_GATE_DB".BUNKER_GATE.HOP_3_MAX_LS;
      );
      =     L 0.0;
      A     L 0.0;
      A     "CC_BUNKER_GATE_DB".BUNKER_GATE.BG_1_DN_LS;
      A     "CC_BUNKER_GATE_DB".BUNKER_GATE.BG_2_DN_LS;
      A     "CC_BUNKER_GATE_DB".BUNKER_GATE.BG_3_DN_LS;
      A     "CC_BUNKER_GATE_DB".BUNKER_GATE.COAL_LD_STP_PB;
      S     "CC_BUNKER_GATE_DB".BUNKER_GATE.COAL_LD_STA_PB_AUTO_SET;
      A     L 0.0;
      FP    "CC_BUNKER_GATE_DB".BUNKER_GATE.PULSE_22;
      R     "CC_BUNKER_GATE_DB".BUNKER_GATE.BG_1_AUTO_DN_CMD_RCHD;
      R     "CC_BUNKER_GATE_DB".BUNKER_GATE.BG_2_AUTO_DN_CMD_RCHD;
      R     "CC_BUNKER_GATE_DB".BUNKER_GATE.BG_3_AUTO_DN_CMD_RCHD;
NETWORK
TITLE = AUTO SEQUENCE INDICATION`
      A     "ALWAYS_ON";
      A(;
      AN    "CC_BUNKER_GATE_DB".BUNKER_GATE.LCS_MD;
      A(;
      A     "CC_BUNKER_GATE_DB".BUNKER_GATE.INTERLOCK_BIT;
      A     "CC_BUNKER_GATE_DB".BUNKER_GATE.SA_MD;
      A(;
      ON    "CC_BUNKER_GATE_DB".BUNKER_GATE.HOP_1_MAX_LS;
      ON    "CC_BUNKER_GATE_DB".BUNKER_GATE.HOP_2_MAX_LS;
      ON    "CC_BUNKER_GATE_DB".BUNKER_GATE.HOP_3_MAX_LS;
      );
      AN    "CC_BUNKER_GATE_DB".BUNKER_GATE.COAL_LD_STA_PB_AUTO_SET;
      O;
      A     "CC_BUNKER_GATE_DB".BUNKER_GATE.COAL_LD_STA_PB_AUTO_SET;
      A     "HALF_SECOND_PULSE_TRAIN";
      );
      O     "MAIN_POWER_DB".LAMP_TEST_PB;
      );
      =     "CC_BUNKER_GATE_DB".BUNKER_GATE.BG_COAL_LD_IND;
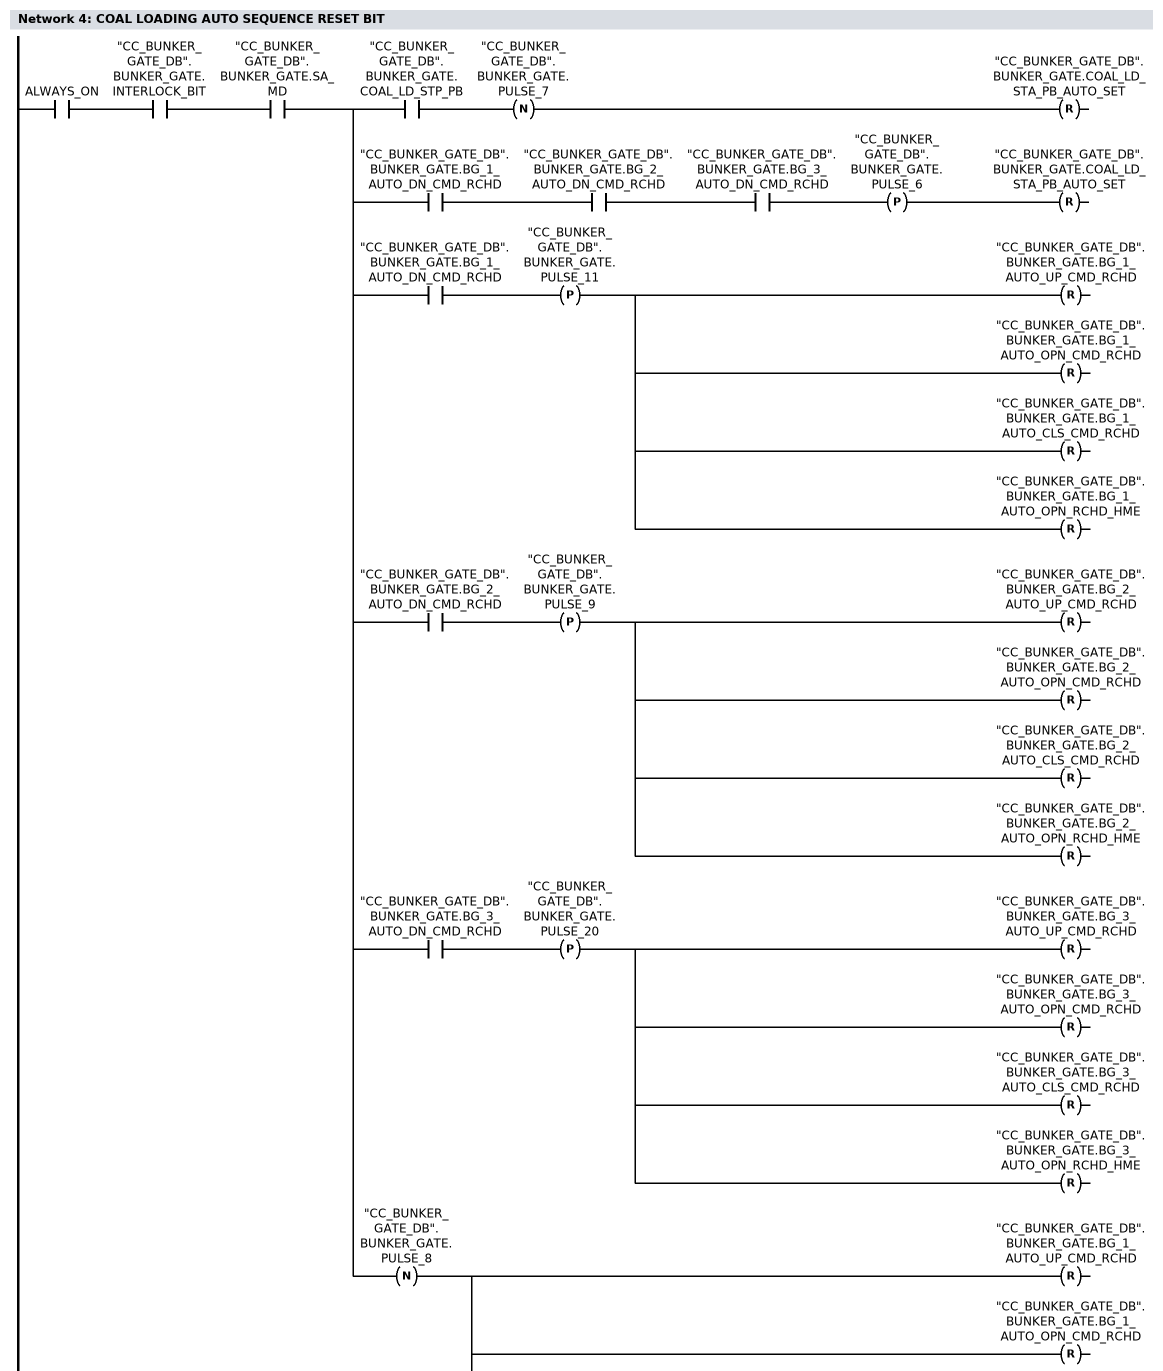
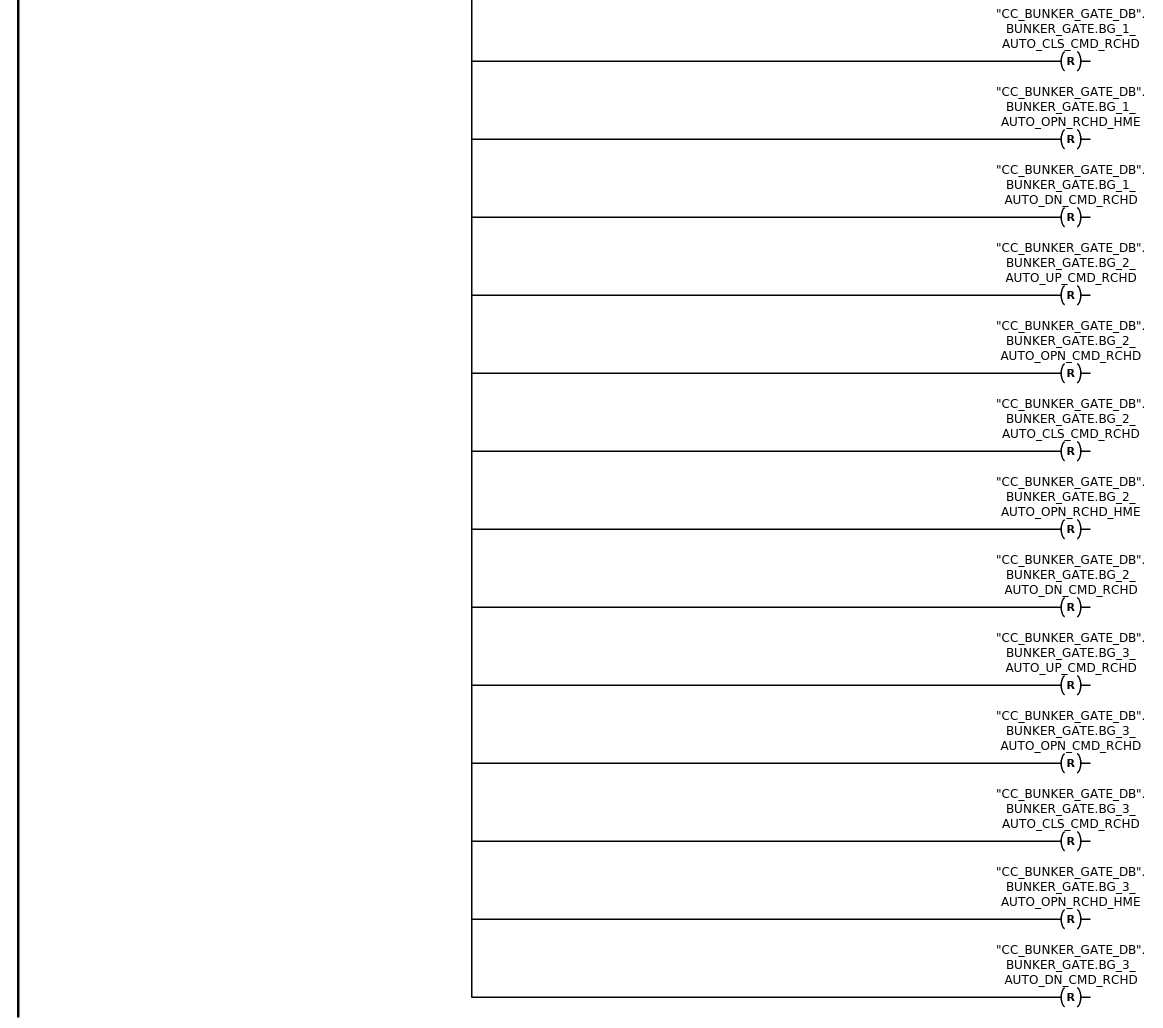
NETWORK
TITLE = COAL LOADING AUTO SEQUENCE RESET BIT
      A     "ALWAYS_ON";
      A     "CC_BUNKER_GATE_DB".BUNKER_GATE.INTERLOCK_BIT;
      A     "CC_BUNKER_GATE_DB".BUNKER_GATE.SA_MD;
      =     L 0.0;
      A     L 0.0;
      A     "CC_BUNKER_GATE_DB".BUNKER_GATE.COAL_LD_STP_PB;
      FN    "CC_BUNKER_GATE_DB".BUNKER_GATE.PULSE_7;
      R     "CC_BUNKER_GATE_DB".BUNKER_GATE.COAL_LD_STA_PB_AUTO_SET;
      A     L 0.0;
      A     "CC_BUNKER_GATE_DB".BUNKER_GATE.BG_1_AUTO_DN_CMD_RCHD;
      A     "CC_BUNKER_GATE_DB".BUNKER_GATE.BG_2_AUTO_DN_CMD_RCHD;
      A     "CC_BUNKER_GATE_DB".BUNKER_GATE.BG_3_AUTO_DN_CMD_RCHD;
      FP    "CC_BUNKER_GATE_DB".BUNKER_GATE.PULSE_6;
      R     "CC_BUNKER_GATE_DB".BUNKER_GATE.COAL_LD_STA_PB_AUTO_SET;
      A     L 0.0;
      A     "CC_BUNKER_GATE_DB".BUNKER_GATE.BG_1_AUTO_DN_CMD_RCHD;
      FP    "CC_BUNKER_GATE_DB".BUNKER_GATE.PULSE_11;
      R     "CC_BUNKER_GATE_DB".BUNKER_GATE.BG_1_AUTO_UP_CMD_RCHD;
      R     "CC_BUNKER_GATE_DB".BUNKER_GATE.BG_1_AUTO_OPN_CMD_RCHD;
      R     "CC_BUNKER_GATE_DB".BUNKER_GATE.BG_1_AUTO_CLS_CMD_RCHD;
      R     "CC_BUNKER_GATE_DB".BUNKER_GATE.BG_1_AUTO_OPN_RCHD_HME;
      A     L 0.0;
      A     "CC_BUNKER_GATE_DB".BUNKER_GATE.BG_2_AUTO_DN_CMD_RCHD;
      FP    "CC_BUNKER_GATE_DB".BUNKER_GATE.PULSE_9;
      R     "CC_BUNKER_GATE_DB".BUNKER_GATE.BG_2_AUTO_UP_CMD_RCHD;
      R     "CC_BUNKER_GATE_DB".BUNKER_GATE.BG_2_AUTO_OPN_CMD_RCHD;
      R     "CC_BUNKER_GATE_DB".BUNKER_GATE.BG_2_AUTO_CLS_CMD_RCHD;
      R     "CC_BUNKER_GATE_DB".BUNKER_GATE.BG_2_AUTO_OPN_RCHD_HME;
      A     L 0.0;
      A     "CC_BUNKER_GATE_DB".BUNKER_GATE.BG_3_AUTO_DN_CMD_RCHD;
      FP    "CC_BUNKER_GATE_DB".BUNKER_GATE.PULSE_20;
      R     "CC_BUNKER_GATE_DB".BUNKER_GATE.BG_3_AUTO_UP_CMD_RCHD;
      R     "CC_BUNKER_GATE_DB".BUNKER_GATE.BG_3_AUTO_OPN_CMD_RCHD;
      R     "CC_BUNKER_GATE_DB".BUNKER_GATE.BG_3_AUTO_CLS_CMD_RCHD;
      R     "CC_BUNKER_GATE_DB".BUNKER_GATE.BG_3_AUTO_OPN_RCHD_HME;
      A     L 0.0;
      FN    "CC_BUNKER_GATE_DB".BUNKER_GATE.PULSE_8;
      R     "CC_BUNKER_GATE_DB".BUNKER_GATE.BG_1_AUTO_UP_CMD_RCHD;
      R     "CC_BUNKER_GATE_DB".BUNKER_GATE.BG_1_AUTO_OPN_CMD_RCHD;
      R     "CC_BUNKER_GATE_DB".BUNKER_GATE.BG_1_AUTO_CLS_CMD_RCHD;
      R     "CC_BUNKER_GATE_DB".BUNKER_GATE.BG_1_AUTO_OPN_RCHD_HME;
      R     "CC_BUNKER_GATE_DB".BUNKER_GATE.BG_1_AUTO_DN_CMD_RCHD;
      R     "CC_BUNKER_GATE_DB".BUNKER_GATE.BG_2_AUTO_UP_CMD_RCHD;
      R     "CC_BUNKER_GATE_DB".BUNKER_GATE.BG_2_AUTO_OPN_CMD_RCHD;
      R     "CC_BUNKER_GATE_DB".BUNKER_GATE.BG_2_AUTO_CLS_CMD_RCHD;
      R     "CC_BUNKER_GATE_DB".BUNKER_GATE.BG_2_AUTO_OPN_RCHD_HME;
      R     "CC_BUNKER_GATE_DB".BUNKER_GATE.BG_2_AUTO_DN_CMD_RCHD;
      R     "CC_BUNKER_GATE_DB".BUNKER_GATE.BG_3_AUTO_UP_CMD_RCHD;
      R     "CC_BUNKER_GATE_DB".BUNKER_GATE.BG_3_AUTO_OPN_CMD_RCHD;
      R     "CC_BUNKER_GATE_DB".BUNKER_GATE.BG_3_AUTO_CLS_CMD_RCHD;
      R     "CC_BUNKER_GATE_DB".BUNKER_GATE.BG_3_AUTO_OPN_RCHD_HME;
      R     "CC_BUNKER_GATE_DB".BUNKER_GATE.BG_3_AUTO_DN_CMD_RCHD;
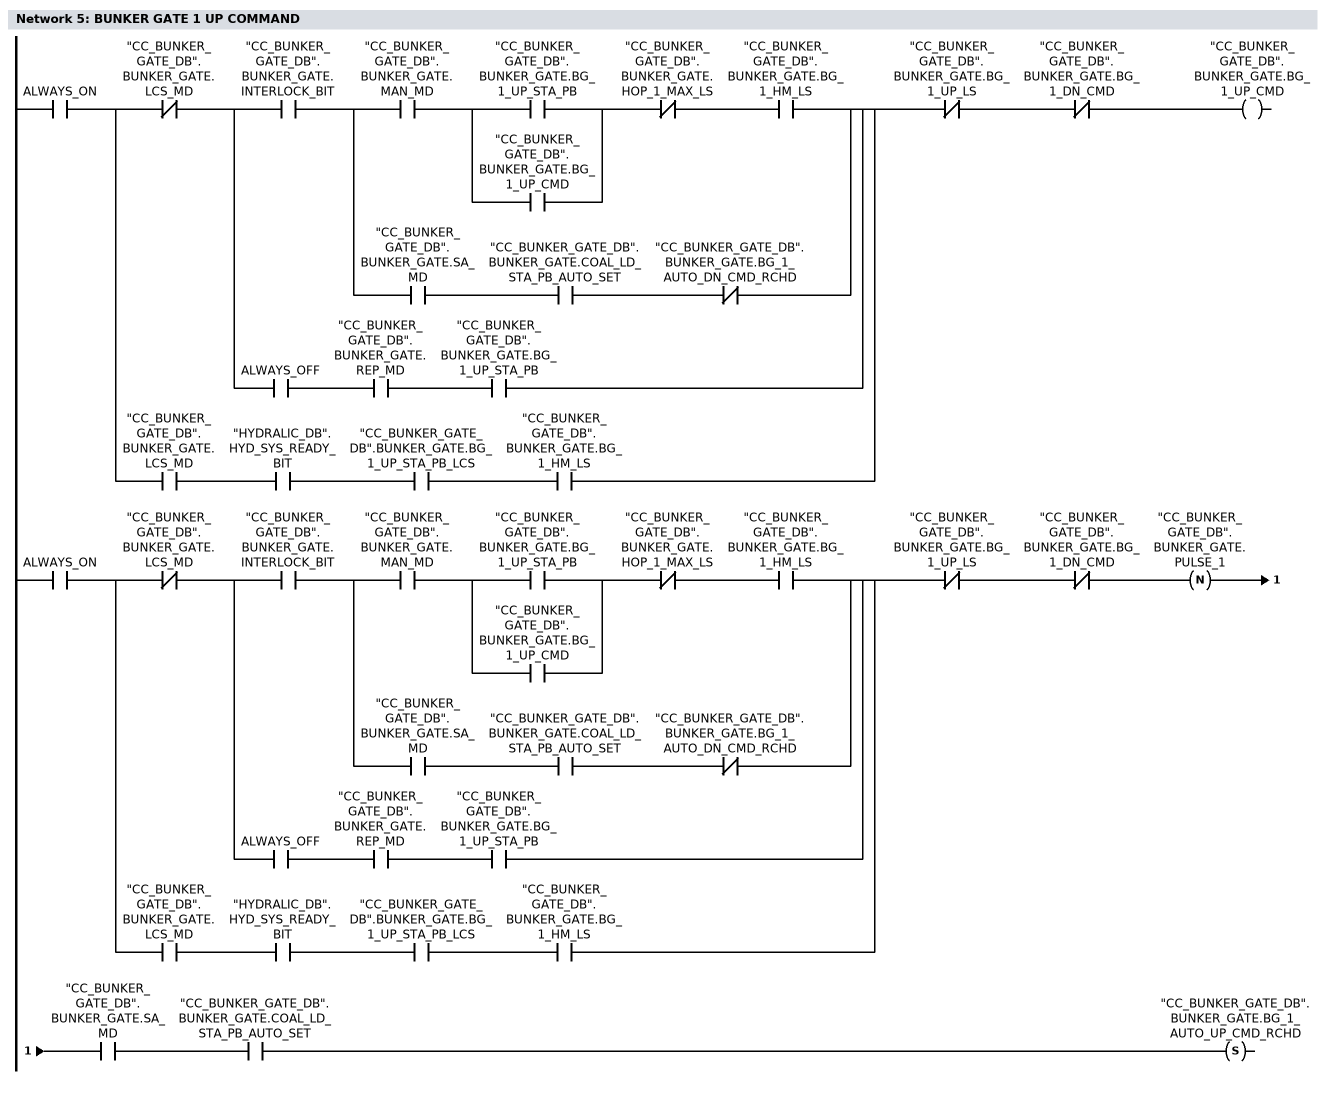
NETWORK
TITLE = BUNKER GATE 1 UP COMMAND
      A     "ALWAYS_ON";
      A(;
      AN    "CC_BUNKER_GATE_DB".BUNKER_GATE.LCS_MD;
      A(;
      A     "CC_BUNKER_GATE_DB".BUNKER_GATE.INTERLOCK_BIT;
      A(;
      A     "CC_BUNKER_GATE_DB".BUNKER_GATE.MAN_MD;
      A(;
      O     "CC_BUNKER_GATE_DB".BUNKER_GATE.BG_1_UP_STA_PB;
      O     "CC_BUNKER_GATE_DB".BUNKER_GATE.BG_1_UP_CMD;
      );
      AN    "CC_BUNKER_GATE_DB".BUNKER_GATE.HOP_1_MAX_LS;
      A     "CC_BUNKER_GATE_DB".BUNKER_GATE.BG_1_HM_LS;
      O;
      A     "CC_BUNKER_GATE_DB".BUNKER_GATE.SA_MD;
      A     "CC_BUNKER_GATE_DB".BUNKER_GATE.COAL_LD_STA_PB_AUTO_SET;
      AN    "CC_BUNKER_GATE_DB".BUNKER_GATE.BG_1_AUTO_DN_CMD_RCHD;
      );
      O;
      A     "ALWAYS_OFF";
      A     "CC_BUNKER_GATE_DB".BUNKER_GATE.REP_MD;
      A     "CC_BUNKER_GATE_DB".BUNKER_GATE.BG_1_UP_STA_PB;
      );
      O;
      A     "CC_BUNKER_GATE_DB".BUNKER_GATE.LCS_MD;
      A     "HYDRALIC_DB".HYD_SYS_READY_BIT;
      A     "CC_BUNKER_GATE_DB".BUNKER_GATE.BG_1_UP_STA_PB_LCS;
      A     "CC_BUNKER_GATE_DB".BUNKER_GATE.BG_1_HM_LS;
      );
      AN    "CC_BUNKER_GATE_DB".BUNKER_GATE.BG_1_UP_LS;
      AN    "CC_BUNKER_GATE_DB".BUNKER_GATE.BG_1_DN_CMD;
      =     L 0.0;
      A     L 0.0;
      BLD   102;
      =     "CC_BUNKER_GATE_DB".BUNKER_GATE.BG_1_UP_CMD;
      A(;
      A     L 0.0;
      FN    "CC_BUNKER_GATE_DB".BUNKER_GATE.PULSE_1;
      );
      A     "CC_BUNKER_GATE_DB".BUNKER_GATE.SA_MD;
      A     "CC_BUNKER_GATE_DB".BUNKER_GATE.COAL_LD_STA_PB_AUTO_SET;
      S     "CC_BUNKER_GATE_DB".BUNKER_GATE.BG_1_AUTO_UP_CMD_RCHD;
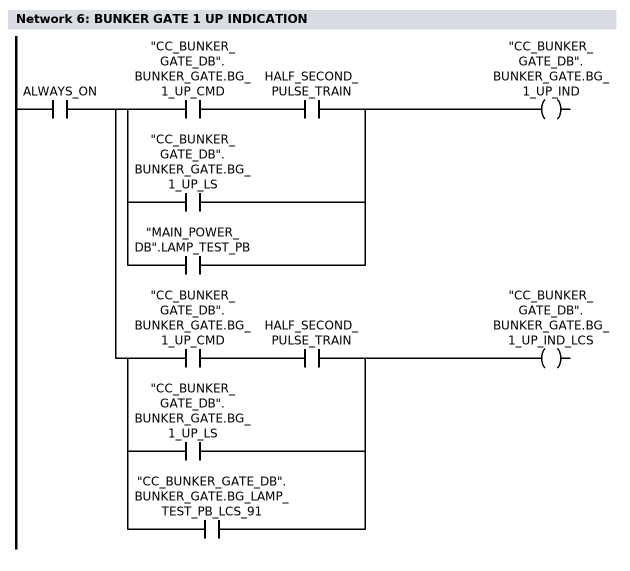
NETWORK
TITLE = BUNKER GATE 1 UP INDICATION
      A     "ALWAYS_ON";
      =     L 0.0;
      A     L 0.0;
      A(;
      A     "CC_BUNKER_GATE_DB".BUNKER_GATE.BG_1_UP_CMD;
      A     "HALF_SECOND_PULSE_TRAIN";
      O     "CC_BUNKER_GATE_DB".BUNKER_GATE.BG_1_UP_LS;
      O     "MAIN_POWER_DB".LAMP_TEST_PB;
      );
      =     "CC_BUNKER_GATE_DB".BUNKER_GATE.BG_1_UP_IND;
      A     L 0.0;
      A(;
      A     "CC_BUNKER_GATE_DB".BUNKER_GATE.BG_1_UP_CMD;
      A     "HALF_SECOND_PULSE_TRAIN";
      O     "CC_BUNKER_GATE_DB".BUNKER_GATE.BG_1_UP_LS;
      O     "CC_BUNKER_GATE_DB".BUNKER_GATE.BG_LAMP_TEST_PB_LCS_91;
      );
      =     "CC_BUNKER_GATE_DB".BUNKER_GATE.BG_1_UP_IND_LCS;
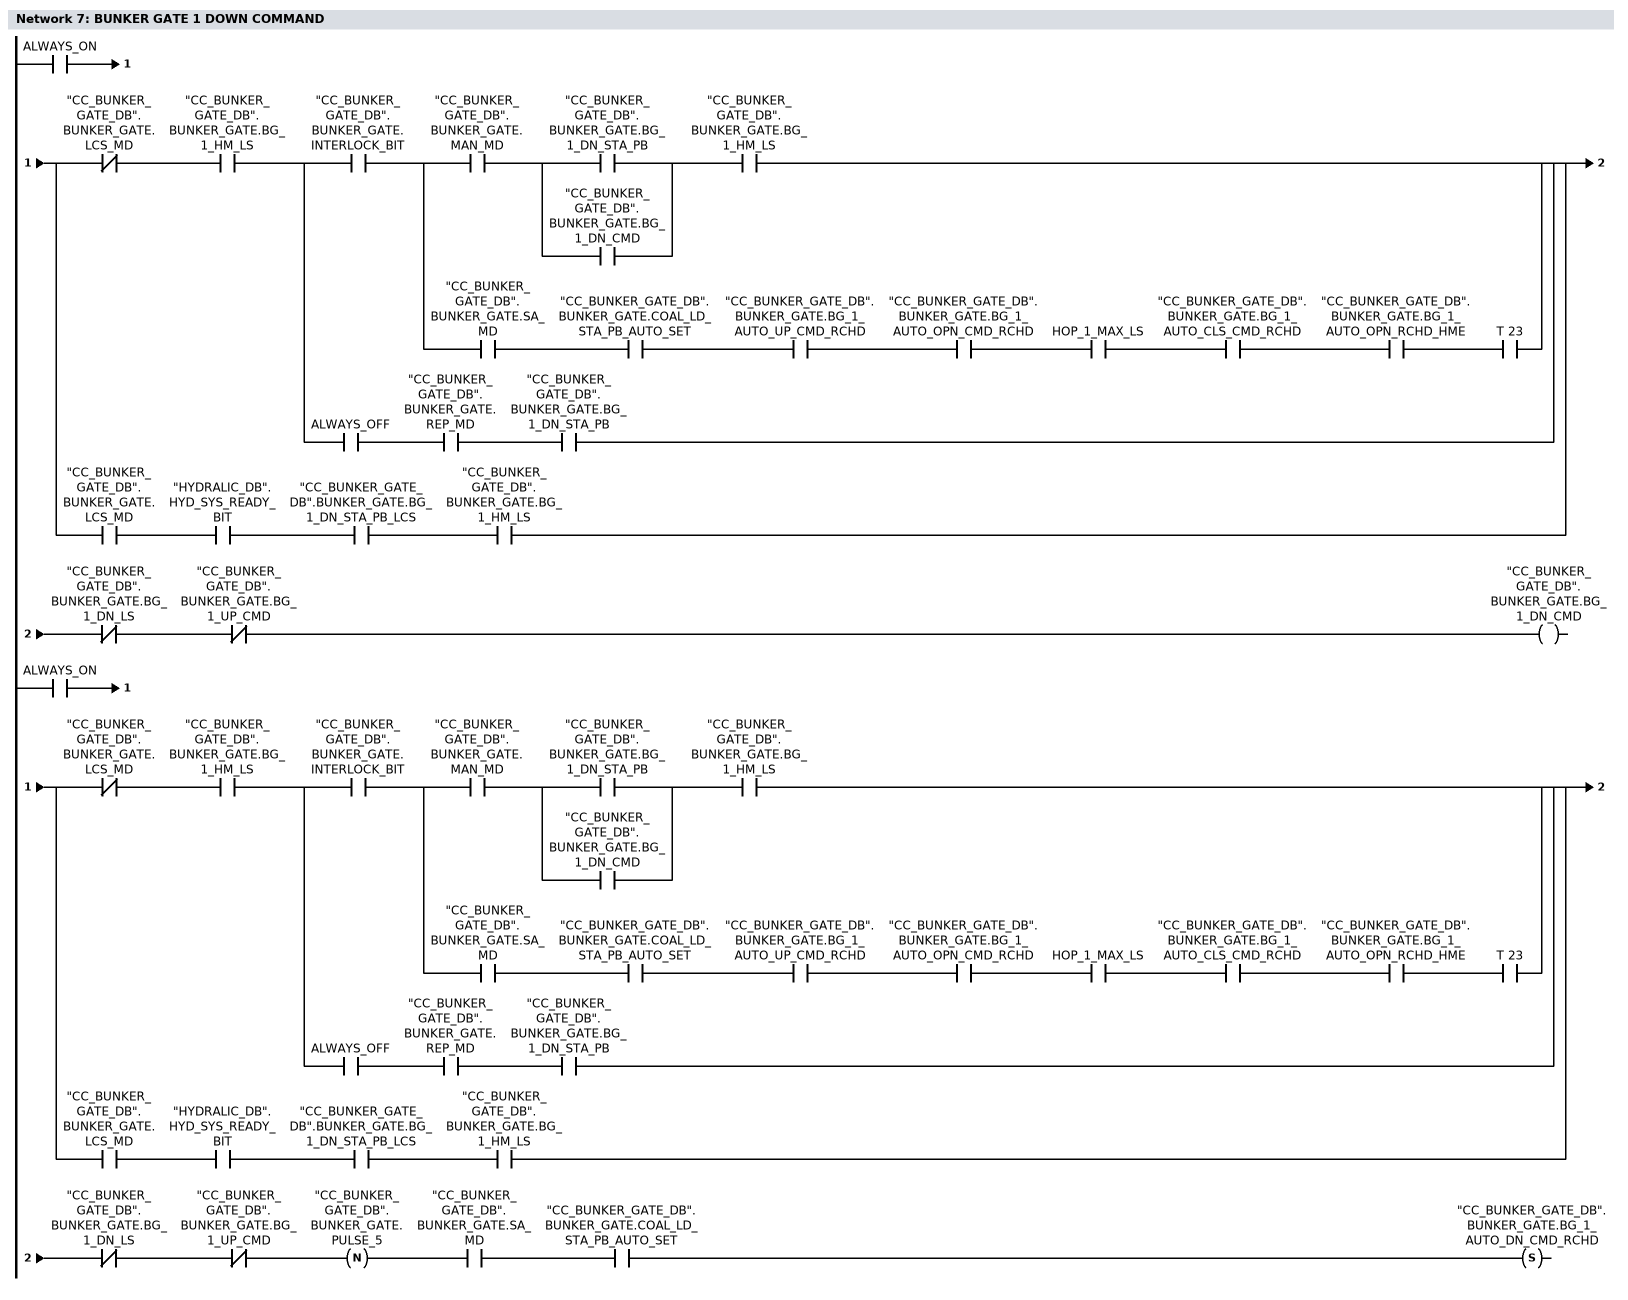
NETWORK
TITLE = BUNKER GATE 1 DOWN COMMAND
      A     "ALWAYS_ON";
      A(;
      AN    "CC_BUNKER_GATE_DB".BUNKER_GATE.LCS_MD;
      A     "CC_BUNKER_GATE_DB".BUNKER_GATE.BG_1_HM_LS;
      A(;
      A     "CC_BUNKER_GATE_DB".BUNKER_GATE.INTERLOCK_BIT;
      A(;
      A     "CC_BUNKER_GATE_DB".BUNKER_GATE.MAN_MD;
      A(;
      O     "CC_BUNKER_GATE_DB".BUNKER_GATE.BG_1_DN_STA_PB;
      O     "CC_BUNKER_GATE_DB".BUNKER_GATE.BG_1_DN_CMD;
      );
      A     "CC_BUNKER_GATE_DB".BUNKER_GATE.BG_1_HM_LS;
      O;
      A     "CC_BUNKER_GATE_DB".BUNKER_GATE.SA_MD;
      A     "CC_BUNKER_GATE_DB".BUNKER_GATE.COAL_LD_STA_PB_AUTO_SET;
      A     "CC_BUNKER_GATE_DB".BUNKER_GATE.BG_1_AUTO_UP_CMD_RCHD;
      A     "CC_BUNKER_GATE_DB".BUNKER_GATE.BG_1_AUTO_OPN_CMD_RCHD;
      A     "HOP_1_MAX_LS";
      A     "CC_BUNKER_GATE_DB".BUNKER_GATE.BG_1_AUTO_CLS_CMD_RCHD;
      A     "CC_BUNKER_GATE_DB".BUNKER_GATE.BG_1_AUTO_OPN_RCHD_HME;
      A     T 23;
      );
      O;
      A     "ALWAYS_OFF";
      A     "CC_BUNKER_GATE_DB".BUNKER_GATE.REP_MD;
      A     "CC_BUNKER_GATE_DB".BUNKER_GATE.BG_1_DN_STA_PB;
      );
      O;
      A     "CC_BUNKER_GATE_DB".BUNKER_GATE.LCS_MD;
      A     "HYDRALIC_DB".HYD_SYS_READY_BIT;
      A     "CC_BUNKER_GATE_DB".BUNKER_GATE.BG_1_DN_STA_PB_LCS;
      A     "CC_BUNKER_GATE_DB".BUNKER_GATE.BG_1_HM_LS;
      );
      AN    "CC_BUNKER_GATE_DB".BUNKER_GATE.BG_1_DN_LS;
      AN    "CC_BUNKER_GATE_DB".BUNKER_GATE.BG_1_UP_CMD;
      =     L 0.0;
      A     L 0.0;
      BLD   102;
      =     "CC_BUNKER_GATE_DB".BUNKER_GATE.BG_1_DN_CMD;
      A(;
      A     L 0.0;
      FN    "CC_BUNKER_GATE_DB".BUNKER_GATE.PULSE_5;
      );
      A     "CC_BUNKER_GATE_DB".BUNKER_GATE.SA_MD;
      A     "CC_BUNKER_GATE_DB".BUNKER_GATE.COAL_LD_STA_PB_AUTO_SET;
      S     "CC_BUNKER_GATE_DB".BUNKER_GATE.BG_1_AUTO_DN_CMD_RCHD;
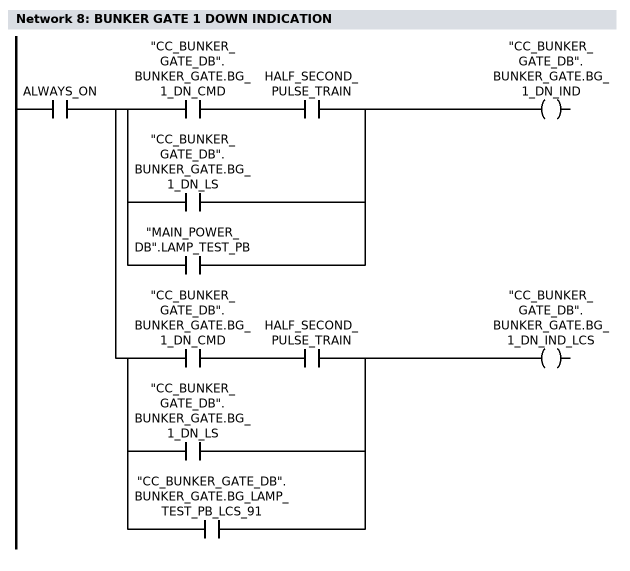
NETWORK
TITLE = BUNKER GATE 1 DOWN INDICATION
      A     "ALWAYS_ON";
      =     L 0.0;
      A     L 0.0;
      A(;
      A     "CC_BUNKER_GATE_DB".BUNKER_GATE.BG_1_DN_CMD;
      A     "HALF_SECOND_PULSE_TRAIN";
      O     "CC_BUNKER_GATE_DB".BUNKER_GATE.BG_1_DN_LS;
      O     "MAIN_POWER_DB".LAMP_TEST_PB;
      );
      =     "CC_BUNKER_GATE_DB".BUNKER_GATE.BG_1_DN_IND;
      A     L 0.0;
      A(;
      A     "CC_BUNKER_GATE_DB".BUNKER_GATE.BG_1_DN_CMD;
      A     "HALF_SECOND_PULSE_TRAIN";
      O     "CC_BUNKER_GATE_DB".BUNKER_GATE.BG_1_DN_LS;
      O     "CC_BUNKER_GATE_DB".BUNKER_GATE.BG_LAMP_TEST_PB_LCS_91;
      );
      =     "CC_BUNKER_GATE_DB".BUNKER_GATE.BG_1_DN_IND_LCS;
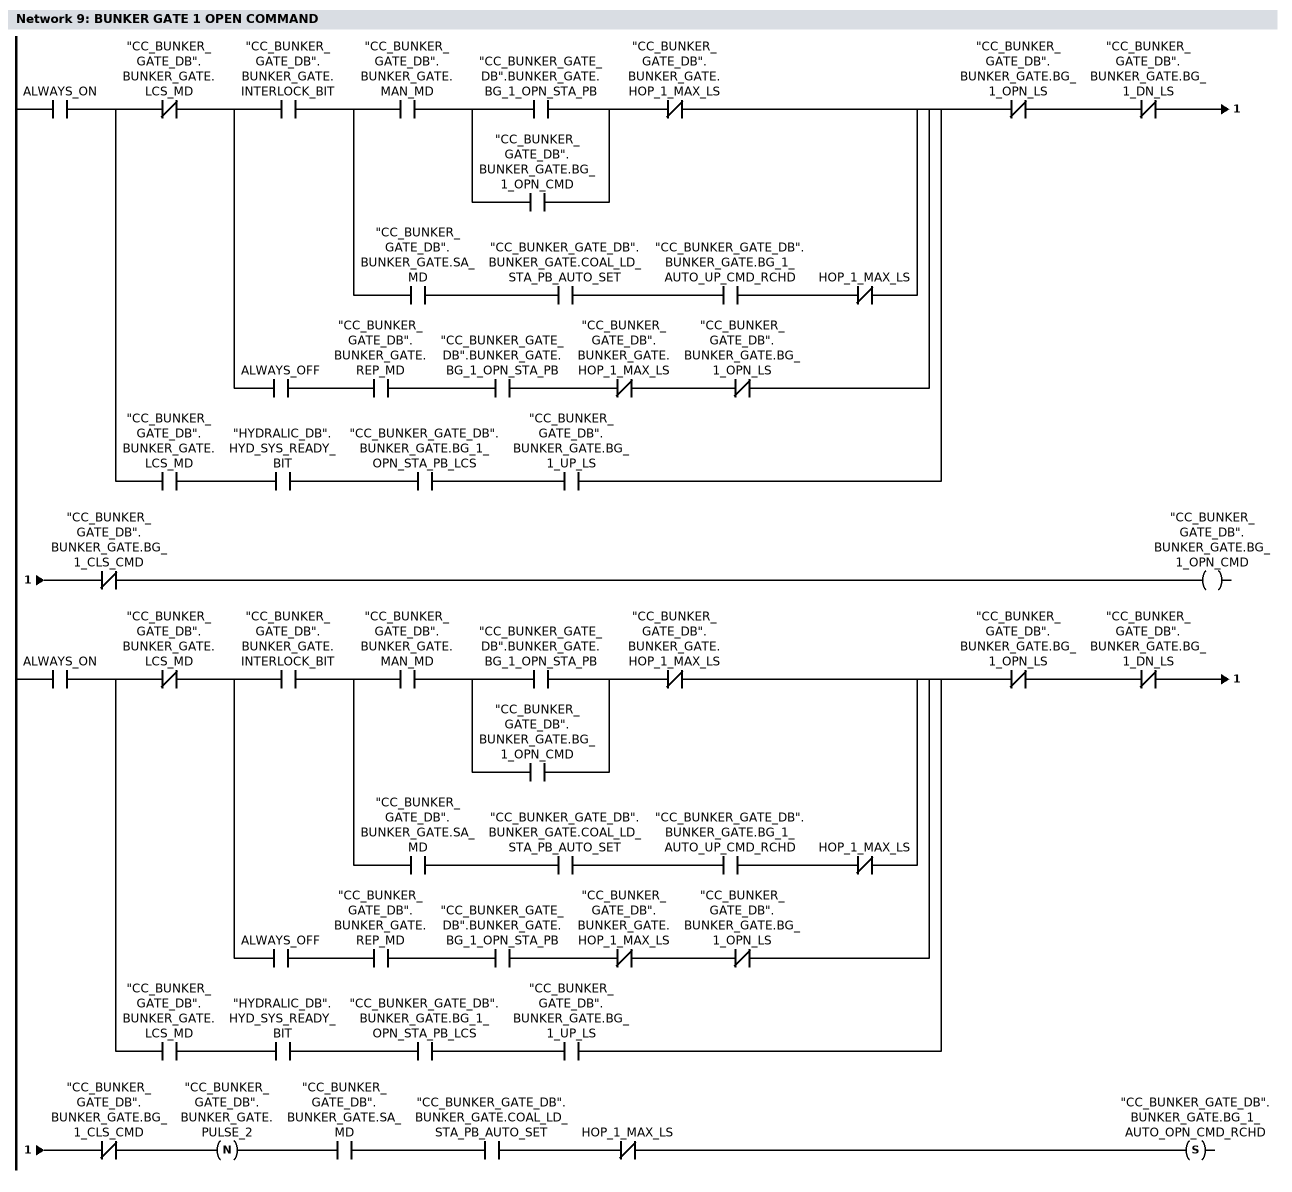
NETWORK
TITLE = BUNKER GATE 1 OPEN COMMAND
      A     "ALWAYS_ON";
      A(;
      AN    "CC_BUNKER_GATE_DB".BUNKER_GATE.LCS_MD;
      A(;
      A     "CC_BUNKER_GATE_DB".BUNKER_GATE.INTERLOCK_BIT;
      A(;
      A     "CC_BUNKER_GATE_DB".BUNKER_GATE.MAN_MD;
      A(;
      O     "CC_BUNKER_GATE_DB".BUNKER_GATE.BG_1_OPN_STA_PB;
      O     "CC_BUNKER_GATE_DB".BUNKER_GATE.BG_1_OPN_CMD;
      );
      AN    "CC_BUNKER_GATE_DB".BUNKER_GATE.HOP_1_MAX_LS;
      O;
      A     "CC_BUNKER_GATE_DB".BUNKER_GATE.SA_MD;
      A     "CC_BUNKER_GATE_DB".BUNKER_GATE.COAL_LD_STA_PB_AUTO_SET;
      A     "CC_BUNKER_GATE_DB".BUNKER_GATE.BG_1_AUTO_UP_CMD_RCHD;
      AN    "HOP_1_MAX_LS";
      );
      O;
      A     "ALWAYS_OFF";
      A     "CC_BUNKER_GATE_DB".BUNKER_GATE.REP_MD;
      A     "CC_BUNKER_GATE_DB".BUNKER_GATE.BG_1_OPN_STA_PB;
      AN    "CC_BUNKER_GATE_DB".BUNKER_GATE.HOP_1_MAX_LS;
      AN    "CC_BUNKER_GATE_DB".BUNKER_GATE.BG_1_OPN_LS;
      );
      O;
      A     "CC_BUNKER_GATE_DB".BUNKER_GATE.LCS_MD;
      A     "HYDRALIC_DB".HYD_SYS_READY_BIT;
      A     "CC_BUNKER_GATE_DB".BUNKER_GATE.BG_1_OPN_STA_PB_LCS;
      A     "CC_BUNKER_GATE_DB".BUNKER_GATE.BG_1_UP_LS;
      );
      AN    "CC_BUNKER_GATE_DB".BUNKER_GATE.BG_1_OPN_LS;
      AN    "CC_BUNKER_GATE_DB".BUNKER_GATE.BG_1_DN_LS;
      AN    "CC_BUNKER_GATE_DB".BUNKER_GATE.BG_1_CLS_CMD;
      =     L 0.0;
      A     L 0.0;
      BLD   102;
      =     "CC_BUNKER_GATE_DB".BUNKER_GATE.BG_1_OPN_CMD;
      A(;
      A     L 0.0;
      FN    "CC_BUNKER_GATE_DB".BUNKER_GATE.PULSE_2;
      );
      A     "CC_BUNKER_GATE_DB".BUNKER_GATE.SA_MD;
      A     "CC_BUNKER_GATE_DB".BUNKER_GATE.COAL_LD_STA_PB_AUTO_SET;
      AN    "HOP_1_MAX_LS";
      S     "CC_BUNKER_GATE_DB".BUNKER_GATE.BG_1_AUTO_OPN_CMD_RCHD;
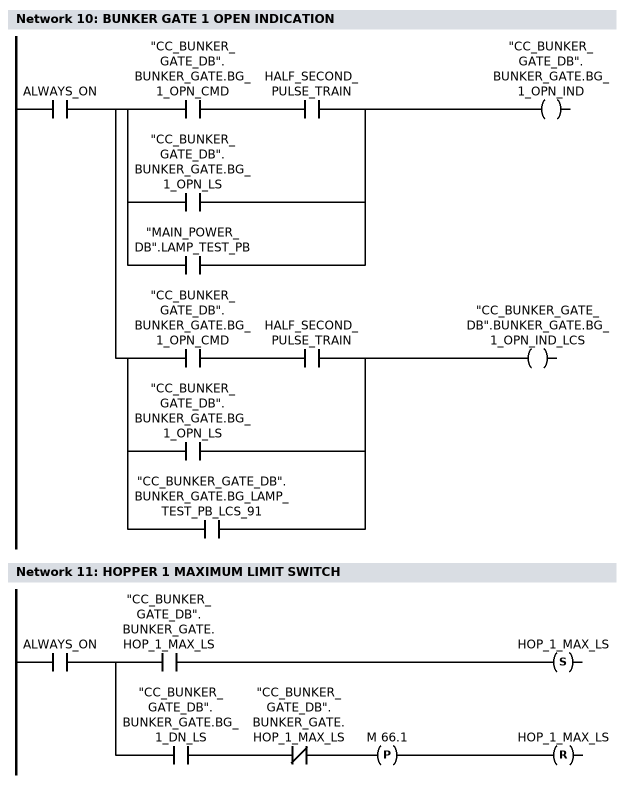
NETWORK
TITLE = BUNKER GATE 1 OPEN INDICATION
      A     "ALWAYS_ON";
      =     L 0.0;
      A     L 0.0;
      A(;
      A     "CC_BUNKER_GATE_DB".BUNKER_GATE.BG_1_OPN_CMD;
      A     "HALF_SECOND_PULSE_TRAIN";
      O     "CC_BUNKER_GATE_DB".BUNKER_GATE.BG_1_OPN_LS;
      O     "MAIN_POWER_DB".LAMP_TEST_PB;
      );
      =     "CC_BUNKER_GATE_DB".BUNKER_GATE.BG_1_OPN_IND;
      A     L 0.0;
      A(;
      A     "CC_BUNKER_GATE_DB".BUNKER_GATE.BG_1_OPN_CMD;
      A     "HALF_SECOND_PULSE_TRAIN";
      O     "CC_BUNKER_GATE_DB".BUNKER_GATE.BG_1_OPN_LS;
      O     "CC_BUNKER_GATE_DB".BUNKER_GATE.BG_LAMP_TEST_PB_LCS_91;
      );
      =     "CC_BUNKER_GATE_DB".BUNKER_GATE.BG_1_OPN_IND_LCS;
NETWORK
TITLE = HOPPER 1 MAXIMUM LIMIT SWITCH
      A     "ALWAYS_ON";
      =     L 0.0;
      A     L 0.0;
      A     "CC_BUNKER_GATE_DB".BUNKER_GATE.HOP_1_MAX_LS;
      S     "HOP_1_MAX_LS";
      A     L 0.0;
      A     "CC_BUNKER_GATE_DB".BUNKER_GATE.BG_1_DN_LS;
      AN    "CC_BUNKER_GATE_DB".BUNKER_GATE.HOP_1_MAX_LS;
      FP    M 66.1;
      R     "HOP_1_MAX_LS";
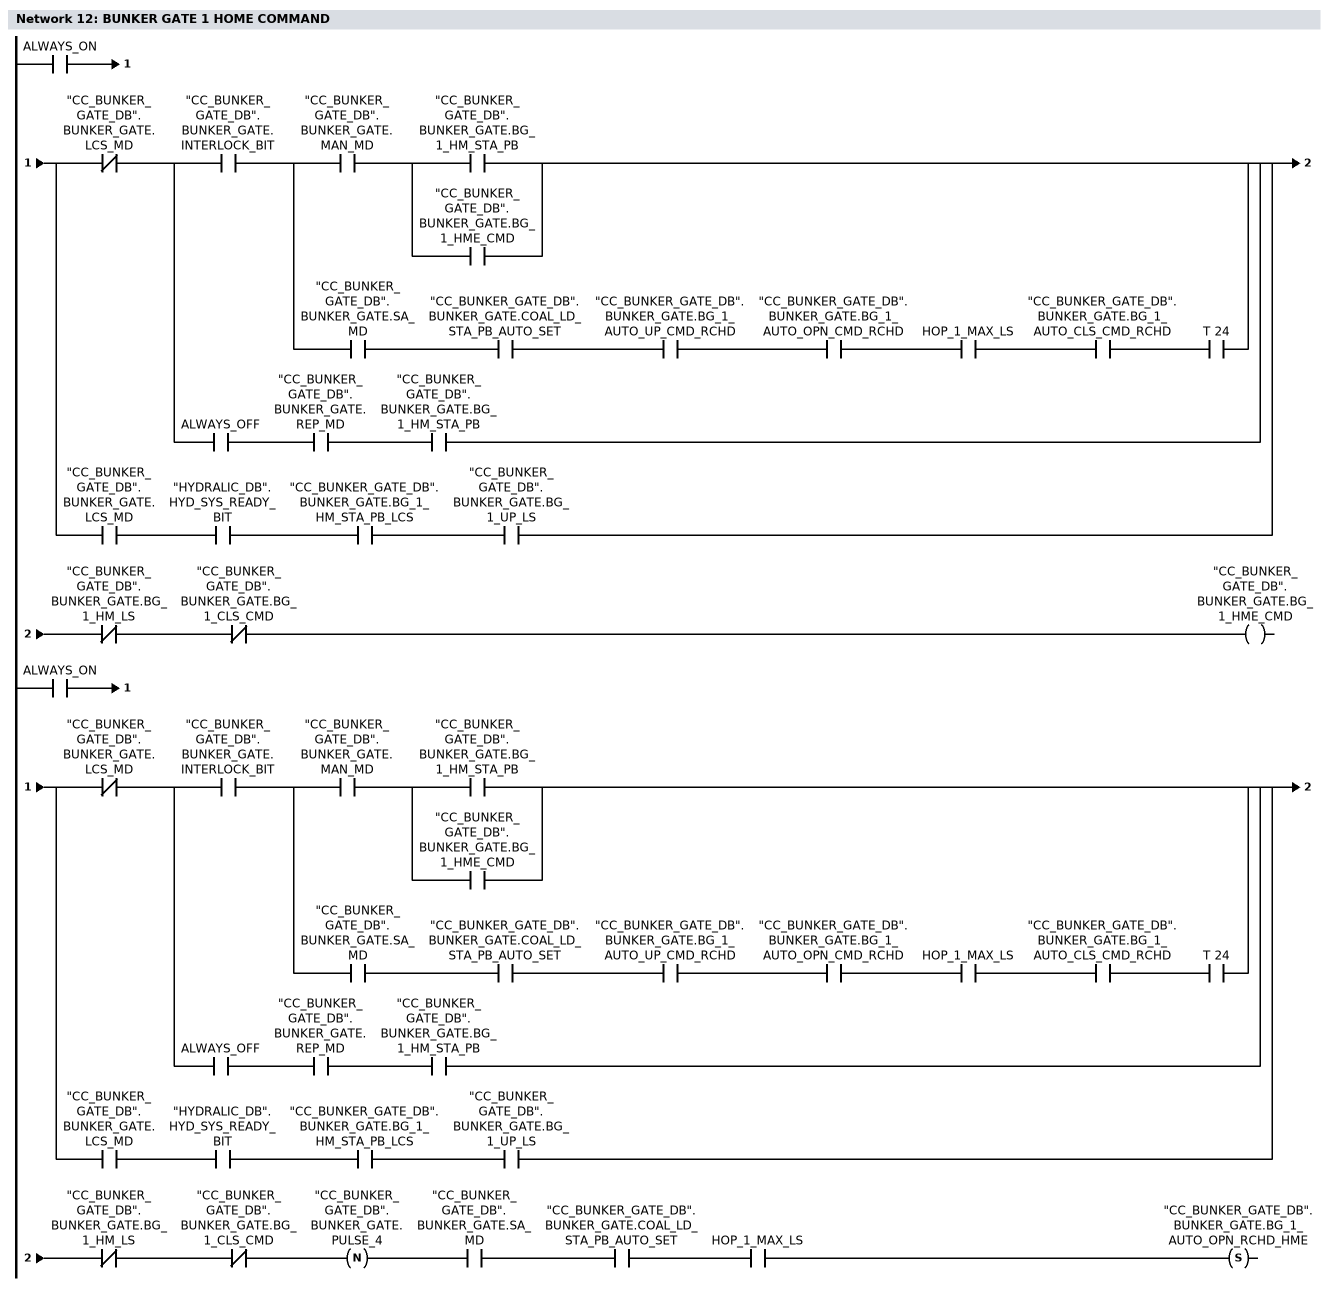
NETWORK
TITLE = BUNKER GATE 1 HOME COMMAND
      A     "ALWAYS_ON";
      A(;
      AN    "CC_BUNKER_GATE_DB".BUNKER_GATE.LCS_MD;
      A(;
      A     "CC_BUNKER_GATE_DB".BUNKER_GATE.INTERLOCK_BIT;
      A(;
      A     "CC_BUNKER_GATE_DB".BUNKER_GATE.MAN_MD;
      A(;
      O     "CC_BUNKER_GATE_DB".BUNKER_GATE.BG_1_HM_STA_PB;
      O     "CC_BUNKER_GATE_DB".BUNKER_GATE.BG_1_HME_CMD;
      );
      O;
      A     "CC_BUNKER_GATE_DB".BUNKER_GATE.SA_MD;
      A     "CC_BUNKER_GATE_DB".BUNKER_GATE.COAL_LD_STA_PB_AUTO_SET;
      A     "CC_BUNKER_GATE_DB".BUNKER_GATE.BG_1_AUTO_UP_CMD_RCHD;
      A     "CC_BUNKER_GATE_DB".BUNKER_GATE.BG_1_AUTO_OPN_CMD_RCHD;
      A     "HOP_1_MAX_LS";
      A     "CC_BUNKER_GATE_DB".BUNKER_GATE.BG_1_AUTO_CLS_CMD_RCHD;
      A     T 24;
      );
      O;
      A     "ALWAYS_OFF";
      A     "CC_BUNKER_GATE_DB".BUNKER_GATE.REP_MD;
      A     "CC_BUNKER_GATE_DB".BUNKER_GATE.BG_1_HM_STA_PB;
      );
      O;
      A     "CC_BUNKER_GATE_DB".BUNKER_GATE.LCS_MD;
      A     "HYDRALIC_DB".HYD_SYS_READY_BIT;
      A     "CC_BUNKER_GATE_DB".BUNKER_GATE.BG_1_HM_STA_PB_LCS;
      A     "CC_BUNKER_GATE_DB".BUNKER_GATE.BG_1_UP_LS;
      );
      AN    "CC_BUNKER_GATE_DB".BUNKER_GATE.BG_1_HM_LS;
      AN    "CC_BUNKER_GATE_DB".BUNKER_GATE.BG_1_CLS_CMD;
      =     L 0.0;
      A     L 0.0;
      BLD   102;
      =     "CC_BUNKER_GATE_DB".BUNKER_GATE.BG_1_HME_CMD;
      A(;
      A     L 0.0;
      FN    "CC_BUNKER_GATE_DB".BUNKER_GATE.PULSE_4;
      );
      A     "CC_BUNKER_GATE_DB".BUNKER_GATE.SA_MD;
      A     "CC_BUNKER_GATE_DB".BUNKER_GATE.COAL_LD_STA_PB_AUTO_SET;
      A     "HOP_1_MAX_LS";
      S     "CC_BUNKER_GATE_DB".BUNKER_GATE.BG_1_AUTO_OPN_RCHD_HME;
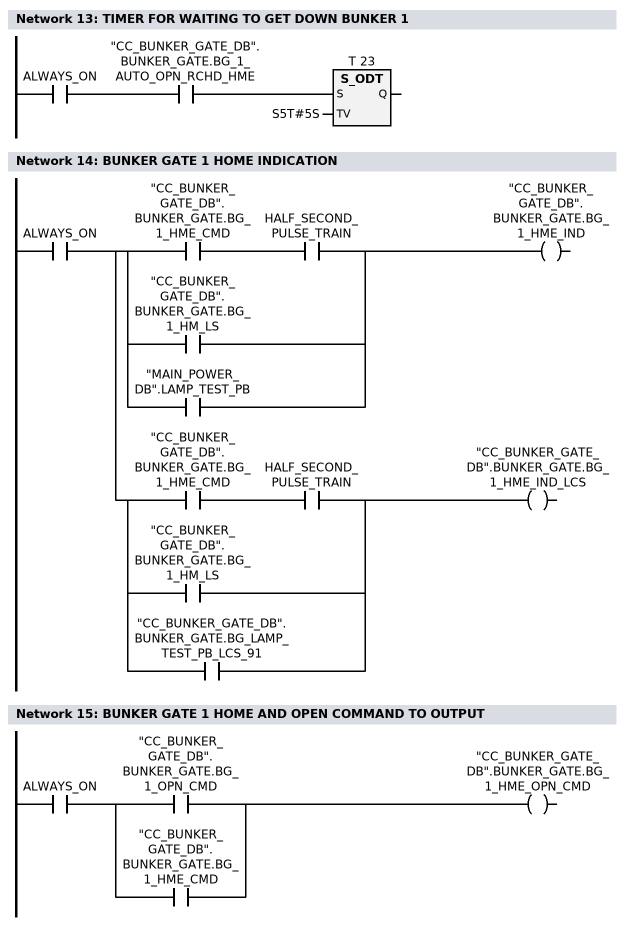
NETWORK
TITLE = TIMER FOR WAITING TO GET DOWN BUNKER 1
      A     "ALWAYS_ON";
      A     "CC_BUNKER_GATE_DB".BUNKER_GATE.BG_1_AUTO_OPN_RCHD_HME;
      L     S5T#5S;
      SD    T 23;
      NOP   0;
      NOP   0;
      NOP   0;
      NOP   0;
NETWORK
TITLE = BUNKER GATE 1 HOME INDICATION
      A     "ALWAYS_ON";
      =     L 0.0;
      A     L 0.0;
      A(;
      A     "CC_BUNKER_GATE_DB".BUNKER_GATE.BG_1_HME_CMD;
      A     "HALF_SECOND_PULSE_TRAIN";
      O     "CC_BUNKER_GATE_DB".BUNKER_GATE.BG_1_HM_LS;
      O     "MAIN_POWER_DB".LAMP_TEST_PB;
      );
      =     "CC_BUNKER_GATE_DB".BUNKER_GATE.BG_1_HME_IND;
      A     L 0.0;
      A(;
      A     "CC_BUNKER_GATE_DB".BUNKER_GATE.BG_1_HME_CMD;
      A     "HALF_SECOND_PULSE_TRAIN";
      O     "CC_BUNKER_GATE_DB".BUNKER_GATE.BG_1_HM_LS;
      O     "CC_BUNKER_GATE_DB".BUNKER_GATE.BG_LAMP_TEST_PB_LCS_91;
      );
      =     "CC_BUNKER_GATE_DB".BUNKER_GATE.BG_1_HME_IND_LCS;
NETWORK
TITLE = BUNKER GATE 1 HOME AND OPEN COMMAND TO OUTPUT
      A     "ALWAYS_ON";
      A(;
      O     "CC_BUNKER_GATE_DB".BUNKER_GATE.BG_1_OPN_CMD;
      O     "CC_BUNKER_GATE_DB".BUNKER_GATE.BG_1_HME_CMD;
      );
      =     "CC_BUNKER_GATE_DB".BUNKER_GATE.BG_1_HME_OPN_CMD;
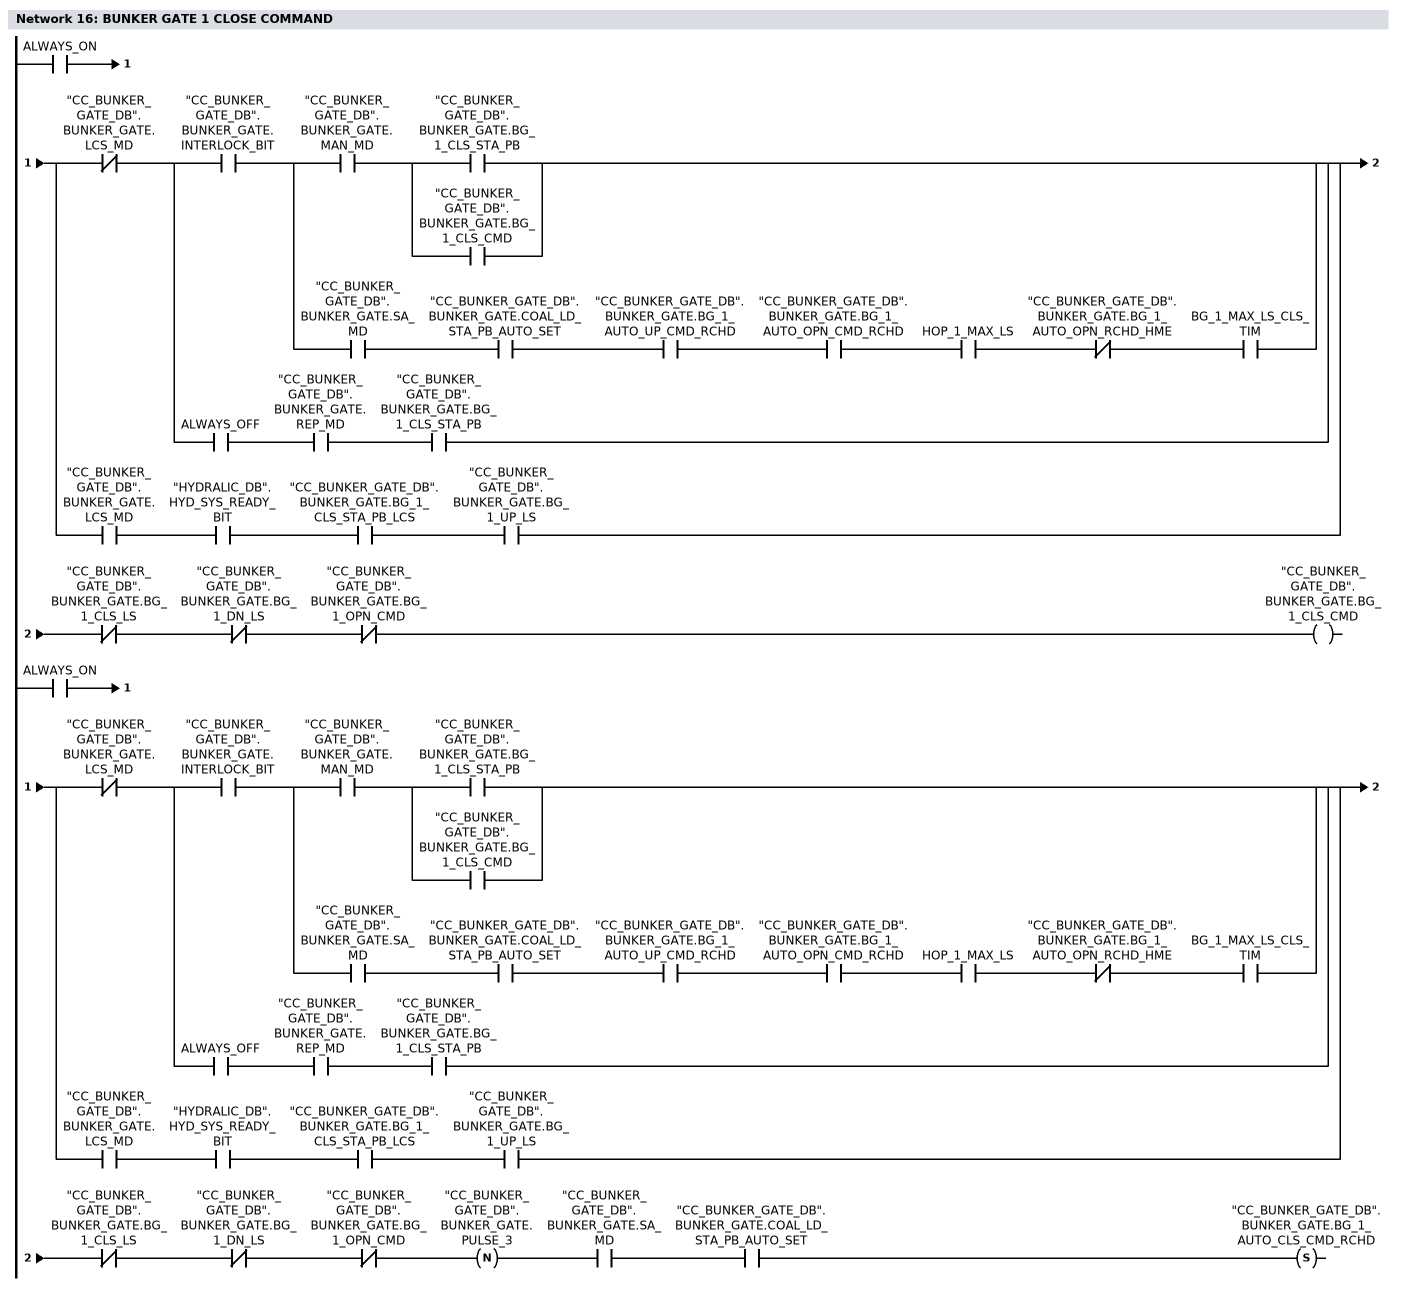
NETWORK
TITLE = BUNKER GATE 1 CLOSE COMMAND
      A     "ALWAYS_ON";
      A(;
      AN    "CC_BUNKER_GATE_DB".BUNKER_GATE.LCS_MD;
      A(;
      A     "CC_BUNKER_GATE_DB".BUNKER_GATE.INTERLOCK_BIT;
      A(;
      A     "CC_BUNKER_GATE_DB".BUNKER_GATE.MAN_MD;
      A(;
      O     "CC_BUNKER_GATE_DB".BUNKER_GATE.BG_1_CLS_STA_PB;
      O     "CC_BUNKER_GATE_DB".BUNKER_GATE.BG_1_CLS_CMD;
      );
      O;
      A     "CC_BUNKER_GATE_DB".BUNKER_GATE.SA_MD;
      A     "CC_BUNKER_GATE_DB".BUNKER_GATE.COAL_LD_STA_PB_AUTO_SET;
      A     "CC_BUNKER_GATE_DB".BUNKER_GATE.BG_1_AUTO_UP_CMD_RCHD;
      A     "CC_BUNKER_GATE_DB".BUNKER_GATE.BG_1_AUTO_OPN_CMD_RCHD;
      A     "HOP_1_MAX_LS";
      AN    "CC_BUNKER_GATE_DB".BUNKER_GATE.BG_1_AUTO_OPN_RCHD_HME;
      A     "BG_1_MAX_LS_CLS_TIM";
      );
      O;
      A     "ALWAYS_OFF";
      A     "CC_BUNKER_GATE_DB".BUNKER_GATE.REP_MD;
      A     "CC_BUNKER_GATE_DB".BUNKER_GATE.BG_1_CLS_STA_PB;
      );
      O;
      A     "CC_BUNKER_GATE_DB".BUNKER_GATE.LCS_MD;
      A     "HYDRALIC_DB".HYD_SYS_READY_BIT;
      A     "CC_BUNKER_GATE_DB".BUNKER_GATE.BG_1_CLS_STA_PB_LCS;
      A     "CC_BUNKER_GATE_DB".BUNKER_GATE.BG_1_UP_LS;
      );
      AN    "CC_BUNKER_GATE_DB".BUNKER_GATE.BG_1_CLS_LS;
      AN    "CC_BUNKER_GATE_DB".BUNKER_GATE.BG_1_DN_LS;
      AN    "CC_BUNKER_GATE_DB".BUNKER_GATE.BG_1_OPN_CMD;
      =     L 0.0;
      A     L 0.0;
      BLD   102;
      =     "CC_BUNKER_GATE_DB".BUNKER_GATE.BG_1_CLS_CMD;
      A(;
      A     L 0.0;
      FN    "CC_BUNKER_GATE_DB".BUNKER_GATE.PULSE_3;
      );
      A     "CC_BUNKER_GATE_DB".BUNKER_GATE.SA_MD;
      A     "CC_BUNKER_GATE_DB".BUNKER_GATE.COAL_LD_STA_PB_AUTO_SET;
      S     "CC_BUNKER_GATE_DB".BUNKER_GATE.BG_1_AUTO_CLS_CMD_RCHD;
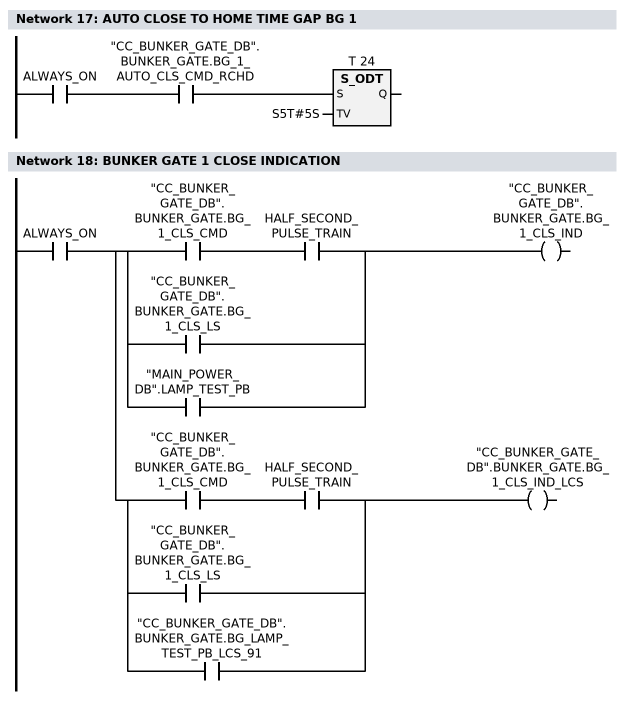
NETWORK
TITLE = AUTO CLOSE TO HOME TIME GAP BG 1
      A     "ALWAYS_ON";
      A     "CC_BUNKER_GATE_DB".BUNKER_GATE.BG_1_AUTO_CLS_CMD_RCHD;
      L     S5T#5S;
      SD    T 24;
      NOP   0;
      NOP   0;
      NOP   0;
      NOP   0;
NETWORK
TITLE = BUNKER GATE 1 CLOSE INDICATION
      A     "ALWAYS_ON";
      =     L 0.0;
      A     L 0.0;
      A(;
      A     "CC_BUNKER_GATE_DB".BUNKER_GATE.BG_1_CLS_CMD;
      A     "HALF_SECOND_PULSE_TRAIN";
      O     "CC_BUNKER_GATE_DB".BUNKER_GATE.BG_1_CLS_LS;
      O     "MAIN_POWER_DB".LAMP_TEST_PB;
      );
      =     "CC_BUNKER_GATE_DB".BUNKER_GATE.BG_1_CLS_IND;
      A     L 0.0;
      A(;
      A     "CC_BUNKER_GATE_DB".BUNKER_GATE.BG_1_CLS_CMD;
      A     "HALF_SECOND_PULSE_TRAIN";
      O     "CC_BUNKER_GATE_DB".BUNKER_GATE.BG_1_CLS_LS;
      O     "CC_BUNKER_GATE_DB".BUNKER_GATE.BG_LAMP_TEST_PB_LCS_91;
      );
      =     "CC_BUNKER_GATE_DB".BUNKER_GATE.BG_1_CLS_IND_LCS;
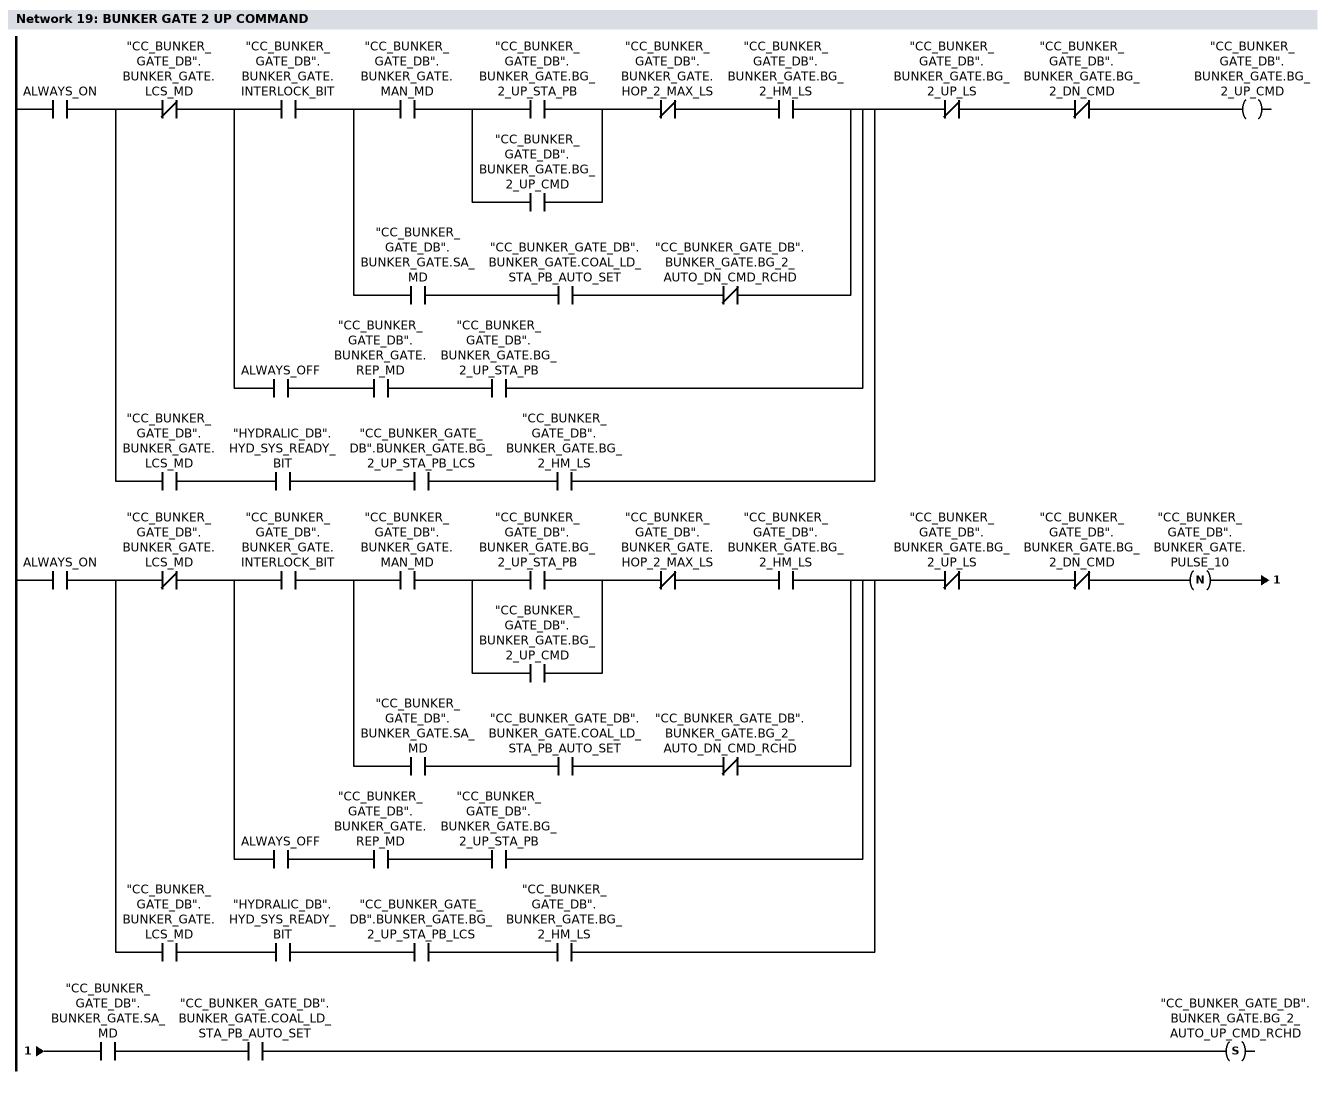
NETWORK
TITLE = BUNKER GATE 2 UP COMMAND
      A     "ALWAYS_ON";
      A(;
      AN    "CC_BUNKER_GATE_DB".BUNKER_GATE.LCS_MD;
      A(;
      A     "CC_BUNKER_GATE_DB".BUNKER_GATE.INTERLOCK_BIT;
      A(;
      A     "CC_BUNKER_GATE_DB".BUNKER_GATE.MAN_MD;
      A(;
      O     "CC_BUNKER_GATE_DB".BUNKER_GATE.BG_2_UP_STA_PB;
      O     "CC_BUNKER_GATE_DB".BUNKER_GATE.BG_2_UP_CMD;
      );
      AN    "CC_BUNKER_GATE_DB".BUNKER_GATE.HOP_2_MAX_LS;
      A     "CC_BUNKER_GATE_DB".BUNKER_GATE.BG_2_HM_LS;
      O;
      A     "CC_BUNKER_GATE_DB".BUNKER_GATE.SA_MD;
      A     "CC_BUNKER_GATE_DB".BUNKER_GATE.COAL_LD_STA_PB_AUTO_SET;
      AN    "CC_BUNKER_GATE_DB".BUNKER_GATE.BG_2_AUTO_DN_CMD_RCHD;
      );
      O;
      A     "ALWAYS_OFF";
      A     "CC_BUNKER_GATE_DB".BUNKER_GATE.REP_MD;
      A     "CC_BUNKER_GATE_DB".BUNKER_GATE.BG_2_UP_STA_PB;
      );
      O;
      A     "CC_BUNKER_GATE_DB".BUNKER_GATE.LCS_MD;
      A     "HYDRALIC_DB".HYD_SYS_READY_BIT;
      A     "CC_BUNKER_GATE_DB".BUNKER_GATE.BG_2_UP_STA_PB_LCS;
      A     "CC_BUNKER_GATE_DB".BUNKER_GATE.BG_2_HM_LS;
      );
      AN    "CC_BUNKER_GATE_DB".BUNKER_GATE.BG_2_UP_LS;
      AN    "CC_BUNKER_GATE_DB".BUNKER_GATE.BG_2_DN_CMD;
      =     L 0.0;
      A     L 0.0;
      BLD   102;
      =     "CC_BUNKER_GATE_DB".BUNKER_GATE.BG_2_UP_CMD;
      A(;
      A     L 0.0;
      FN    "CC_BUNKER_GATE_DB".BUNKER_GATE.PULSE_10;
      );
      A     "CC_BUNKER_GATE_DB".BUNKER_GATE.SA_MD;
      A     "CC_BUNKER_GATE_DB".BUNKER_GATE.COAL_LD_STA_PB_AUTO_SET;
      S     "CC_BUNKER_GATE_DB".BUNKER_GATE.BG_2_AUTO_UP_CMD_RCHD;
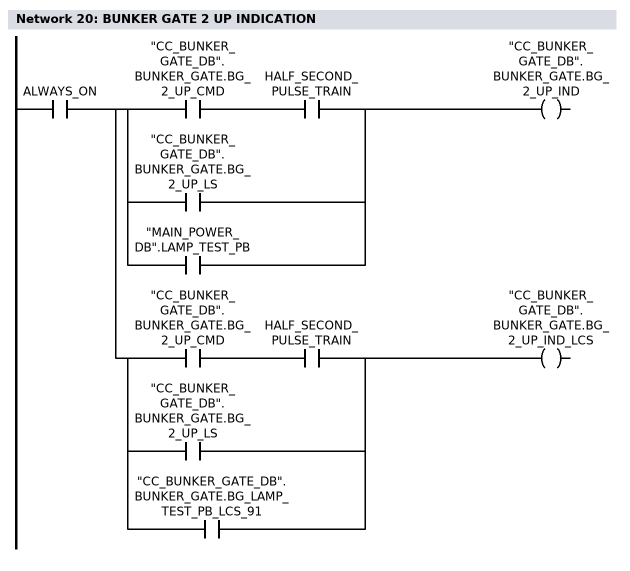
NETWORK
TITLE = BUNKER GATE 2 UP INDICATION
      A     "ALWAYS_ON";
      =     L 0.0;
      A     L 0.0;
      A(;
      A     "CC_BUNKER_GATE_DB".BUNKER_GATE.BG_2_UP_CMD;
      A     "HALF_SECOND_PULSE_TRAIN";
      O     "CC_BUNKER_GATE_DB".BUNKER_GATE.BG_2_UP_LS;
      O     "MAIN_POWER_DB".LAMP_TEST_PB;
      );
      =     "CC_BUNKER_GATE_DB".BUNKER_GATE.BG_2_UP_IND;
      A     L 0.0;
      A(;
      A     "CC_BUNKER_GATE_DB".BUNKER_GATE.BG_2_UP_CMD;
      A     "HALF_SECOND_PULSE_TRAIN";
      O     "CC_BUNKER_GATE_DB".BUNKER_GATE.BG_2_UP_LS;
      O     "CC_BUNKER_GATE_DB".BUNKER_GATE.BG_LAMP_TEST_PB_LCS_91;
      );
      =     "CC_BUNKER_GATE_DB".BUNKER_GATE.BG_2_UP_IND_LCS;
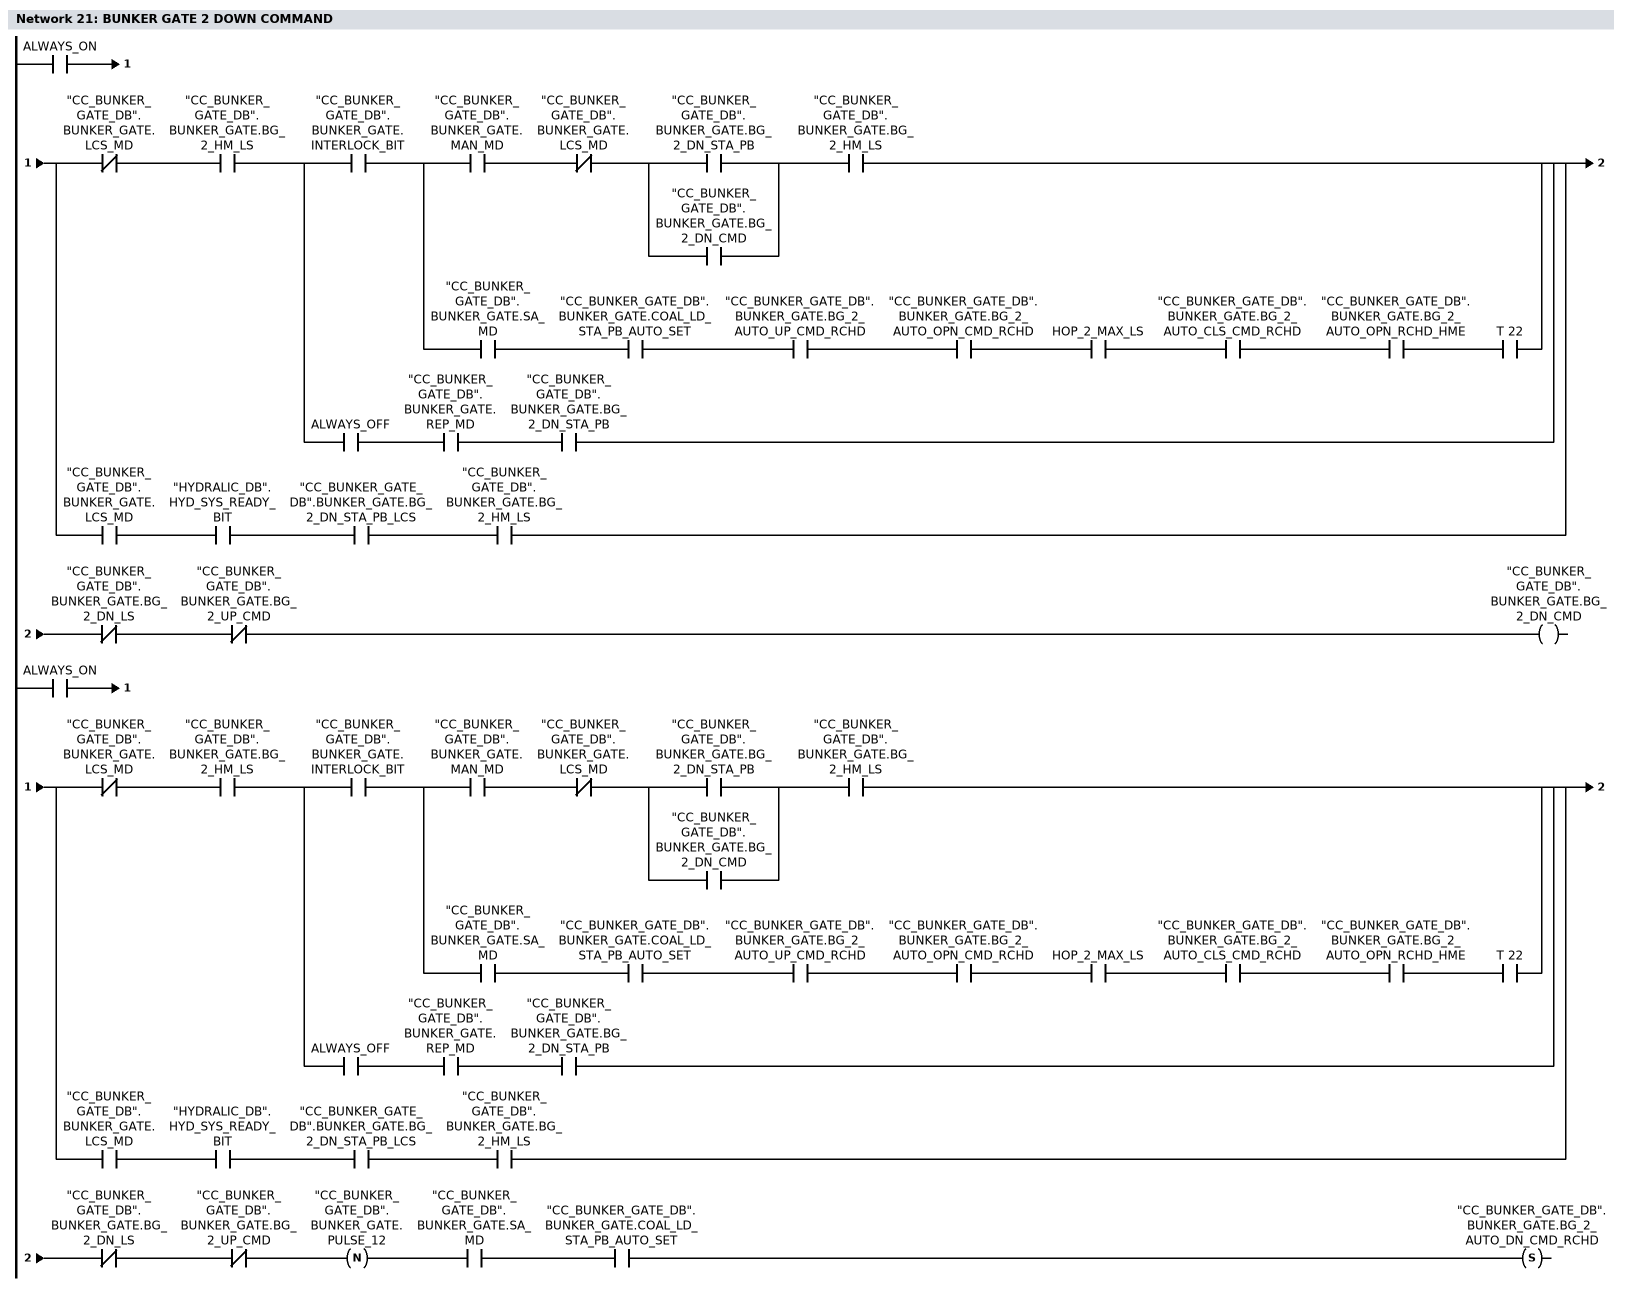
NETWORK
TITLE = BUNKER GATE 2 DOWN COMMAND
      A     "ALWAYS_ON";
      A(;
      AN    "CC_BUNKER_GATE_DB".BUNKER_GATE.LCS_MD;
      A     "CC_BUNKER_GATE_DB".BUNKER_GATE.BG_2_HM_LS;
      A(;
      A     "CC_BUNKER_GATE_DB".BUNKER_GATE.INTERLOCK_BIT;
      A(;
      A     "CC_BUNKER_GATE_DB".BUNKER_GATE.MAN_MD;
      AN    "CC_BUNKER_GATE_DB".BUNKER_GATE.LCS_MD;
      A(;
      O     "CC_BUNKER_GATE_DB".BUNKER_GATE.BG_2_DN_STA_PB;
      O     "CC_BUNKER_GATE_DB".BUNKER_GATE.BG_2_DN_CMD;
      );
      A     "CC_BUNKER_GATE_DB".BUNKER_GATE.BG_2_HM_LS;
      O;
      A     "CC_BUNKER_GATE_DB".BUNKER_GATE.SA_MD;
      A     "CC_BUNKER_GATE_DB".BUNKER_GATE.COAL_LD_STA_PB_AUTO_SET;
      A     "CC_BUNKER_GATE_DB".BUNKER_GATE.BG_2_AUTO_UP_CMD_RCHD;
      A     "CC_BUNKER_GATE_DB".BUNKER_GATE.BG_2_AUTO_OPN_CMD_RCHD;
      A     "HOP_2_MAX_LS";
      A     "CC_BUNKER_GATE_DB".BUNKER_GATE.BG_2_AUTO_CLS_CMD_RCHD;
      A     "CC_BUNKER_GATE_DB".BUNKER_GATE.BG_2_AUTO_OPN_RCHD_HME;
      A     T 22;
      );
      O;
      A     "ALWAYS_OFF";
      A     "CC_BUNKER_GATE_DB".BUNKER_GATE.REP_MD;
      A     "CC_BUNKER_GATE_DB".BUNKER_GATE.BG_2_DN_STA_PB;
      );
      O;
      A     "CC_BUNKER_GATE_DB".BUNKER_GATE.LCS_MD;
      A     "HYDRALIC_DB".HYD_SYS_READY_BIT;
      A     "CC_BUNKER_GATE_DB".BUNKER_GATE.BG_2_DN_STA_PB_LCS;
      A     "CC_BUNKER_GATE_DB".BUNKER_GATE.BG_2_HM_LS;
      );
      AN    "CC_BUNKER_GATE_DB".BUNKER_GATE.BG_2_DN_LS;
      AN    "CC_BUNKER_GATE_DB".BUNKER_GATE.BG_2_UP_CMD;
      =     L 0.0;
      A     L 0.0;
      BLD   102;
      =     "CC_BUNKER_GATE_DB".BUNKER_GATE.BG_2_DN_CMD;
      A(;
      A     L 0.0;
      FN    "CC_BUNKER_GATE_DB".BUNKER_GATE.PULSE_12;
      );
      A     "CC_BUNKER_GATE_DB".BUNKER_GATE.SA_MD;
      A     "CC_BUNKER_GATE_DB".BUNKER_GATE.COAL_LD_STA_PB_AUTO_SET;
      S     "CC_BUNKER_GATE_DB".BUNKER_GATE.BG_2_AUTO_DN_CMD_RCHD;
